LIN {X 0,Y 474.637,Z 227.855,A -85,B 0,C 180,E1 -7347.785,E2 -7347.785} C_VEL
LIN {X 0,Y 474.608,Z 227.868,A -85,B 0,C 180,E1 -7350.888,E2 -7350.888} C_VEL
LIN {X 0,Y 474.599,Z 227.864,A -85,B 0,C 180,E1 -7353.622,E2 -7353.622} C_VEL
LIN {X 0,Y 474.643,Z 227.855,A -85,B 0,C 180,E1 -7356.64,E2 -7356.64} C_VEL
LIN {X 0,Y 474.662,Z 227.851,A -85,B 0,C 180,E1 -7360.087,E2 -7360.087} C_VEL
LIN {X 0,Y 474.645,Z 227.858,A -85,B 0,C 180,E1 -7362.771,E2 -7362.771} C_VEL
LIN {X 0,Y 474.652,Z 227.858,A -85,B 0,C 180,E1 -7365.418,E2 -7365.418} C_VEL
LIN {X 0,Y 474.71,Z 227.848,A -85,B 0,C 180,E1 -7368.034,E2 -7368.034} C_VEL
LIN {X 0,Y 474.707,Z 227.853,A -85,B 0,C 180,E1 -7371.483,E2 -7371.483} C_VEL
LIN {X 0,Y 474.762,Z 227.845,A -85,B 0,C 180,E1 -7374.049,E2 -7374.049} C_VEL
LIN {X 0,Y 474.884,Z 227.829,A -85,B 0,C 180,E1 -7377.452,E2 -7377.452} C_VEL
LIN {X 0,Y 474.91,Z 227.829,A -85,B 0,C 180,E1 -7379.996,E2 -7379.996} C_VEL
LIN {X 0,Y 474.884,Z 227.825,A -85,B 0,C 180,E1 -7382.541,E2 -7382.541} C_VEL
LIN {X 0,Y 474.755,Z 227.847,A -85,B 0,C 180,E1 -7385.944,E2 -7385.944} C_VEL
LIN {X 0,Y 474.708,Z 227.856,A -85,B 0,C 180,E1 -7388.51,E2 -7388.51} C_VEL
LIN {X 0,Y 474.698,Z 227.848,A -85,B 0,C 180,E1 -7391.958,E2 -7391.958} C_VEL
LIN {X 0,Y 474.691,Z 227.848,A -85,B 0,C 180,E1 -7395.451,E2 -7395.451} C_VEL
LIN {X 0,Y 474.652,Z 227.86,A -85,B 0,C 180,E1 -7399.006,E2 -7399.006} C_VEL
LIN {X 0,Y 474.579,Z 227.863,A -85,B 0,C 180,E1 -7401.724,E2 -7401.724} C_VEL
LIN {X 0,Y 474.643,Z 227.86,A -85,B 0,C 180,E1 -7404.488,E2 -7404.488} C_VEL
LIN {X 0,Y 474.681,Z 227.856,A -85,B 0,C 180,E1 -7407.334,E2 -7407.334} C_VEL
LIN {X 0,Y 474.583,Z 227.865,A -85,B 0,C 180,E1 -7410.806,E2 -7410.806} C_VEL
LIN {X 0,Y 474.614,Z 227.86,A -85,B 0,C 180,E1 -7413.979,E2 -7413.979} C_VEL
LIN {X 0,Y 474.551,Z 227.872,A -85,B 0,C 180,E1 -7416.896,E2 -7416.896} C_VEL
LIN {X 0,Y 474.639,Z 227.864,A -85,B 0,C 180,E1 -7419.649,E2 -7419.649} C_VEL
LIN {X 0,Y 474.621,Z 227.863,A -85,B 0,C 180,E1 -7422.926,E2 -7422.926} C_VEL
LIN {X 0,Y 474.585,Z 227.871,A -85,B 0,C 180,E1 -7425.892,E2 -7425.892} C_VEL
LIN {X 0,Y 474.641,Z 227.863,A -85,B 0,C 180,E1 -7429.03,E2 -7429.03} C_VEL
LIN {X 0,Y 474.664,Z 228.034,A -85,B 0,C 180,E1 -7429.413,E2 -7429.413} C_VEL
LIN {X 0,Y 476.042,Z 236.042,A -85,B 0,C 180,E1 -7431.082,E2 -7431.082} C_VEL
LIN {X 0,Y 475.687,Z 249.987,A -85,B 0,C 180,E1 -7433.774,E2 -7433.774} C_VEL
LIN {X 0,Y 475.438,Z 257.892,A -85,B 0,C 180,E1 -7435.224,E2 -7435.224} C_VEL
LIN {X 0,Y 478.234,Z 273.822,A -85,B 0,C 180,E1 -7435.606,E2 -7435.606} C_VEL
LIN {X 0,Y 477.459,Z 365.537,A -85,B 0,C 180,E1 -7437.025,E2 -7437.025} C_VEL
LIN {X 0,Y 477.168,Z 379.142,A -85,B 0,C 180,E1 -7437.417,E2 -7437.417} C_VEL
LIN {X 0,Y 477.152,Z 379.469,A -85,B 0,C 180,E1 -7437.429,E2 -7437.429} C_VEL
LIN {X 0,Y 476.275,Z 385.106,A -85,B 0,C 180,E1 -7437.621,E2 -7437.621} C_VEL
LIN {X 0,Y 473.236,Z 394.135,A -85,B 0,C 180,E1 -7437.957,E2 -7437.957} C_VEL
LIN {X 0,Y 470.185,Z 402.828,A -85,B 0,C 180,E1 -7438.392,E2 -7438.392} C_VEL
LIN {X 0,Y 469.29,Z 407.927,A -85,B 0,C 180,E1 -7438.735,E2 -7438.735} C_VEL
LIN {X 0,Y 468.72,Z 419.724,A -85,B 0,C 180,E1 -7439.723,E2 -7439.723} C_VEL
LIN {X 0,Y 468.195,Z 430.121,A -85,B 0,C 180,E1 -7440.818,E2 -7440.818} C_VEL
LIN {X 0,Y 467.739,Z 439.1,A -85,B 0,C 180,E1 -7441.995,E2 -7441.995} C_VEL
LIN {X 0,Y 467.345,Z 446.512,A -85,B 0,C 180,E1 -7443.183,E2 -7443.183} C_VEL
LIN {X 0,Y 467.063,Z 453.262,A -85,B 0,C 180,E1 -7444.518,E2 -7444.518} C_VEL
LIN {X 0,Y 466.854,Z 459.174,A -85,B 0,C 180,E1 -7446.017,E2 -7446.017} C_VEL
LIN {X 0,Y 466.701,Z 463.326,A -85,B 0,C 180,E1 -7447.418,E2 -7447.418} C_VEL
LIN {X 0,Y 466.582,Z 466.653,A -85,B 0,C 180,E1 -7449.032,E2 -7449.032} C_VEL
LIN {X 0,Y 466.545,Z 468.549,A -85,B 0,C 180,E1 -7450.646,E2 -7450.646} C_VEL
LIN {X 0,Y 466.52,Z 468.981,A -85,B 0,C 180,E1 -7451.616,E2 -7451.616} C_VEL
LIN {X 0,Y 466.521,Z 468.971,A -85,B 0,C 180,E1 -7452.464,E2 -7452.464} C_VEL
LIN {X 0,Y 466.514,Z 468.561,A -85,B 0,C 180,E1 -7453.367,E2 -7453.367} C_VEL
LIN {X 0,Y 466.59,Z 467.307,A -85,B 0,C 180,E1 -7454.555,E2 -7454.555} C_VEL
LIN {X 0,Y 466.641,Z 464.653,A -85,B 0,C 180,E1 -7456.056,E2 -7456.056} C_VEL
LIN {X 0,Y 466.745,Z 461.18,A -85,B 0,C 180,E1 -7457.389,E2 -7457.389} C_VEL
LIN {X 0,Y 466.934,Z 456.593,A -85,B 0,C 180,E1 -7458.716,E2 -7458.716} C_VEL
LIN {X 0,Y 467.209,Z 449.631,A -85,B 0,C 180,E1 -7460.257,E2 -7460.257} C_VEL
LIN {X 0,Y 467.548,Z 442.094,A -85,B 0,C 180,E1 -7461.572,E2 -7461.572} C_VEL
LIN {X 0,Y 467.973,Z 433.15,A -85,B 0,C 180,E1 -7462.826,E2 -7462.826} C_VEL
LIN {X 0,Y 468.408,Z 422.966,A -85,B 0,C 180,E1 -7463.971,E2 -7463.971} C_VEL
LIN {X 0,Y 468.96,Z 412.135,A -85,B 0,C 180,E1 -7464.949,E2 -7464.949} C_VEL
LIN {X 0,Y 469.409,Z 401.596,A -85,B 0,C 180,E1 -7465.707,E2 -7465.707} C_VEL
LIN {X 0,Y 469.91,Z 388.899,A -85,B 0,C 180,E1 -7466.409,E2 -7466.409} C_VEL
LIN {X 0,Y 470.236,Z 376.257,A -85,B 0,C 180,E1 -7466.921,E2 -7466.921} C_VEL
LIN {X 0,Y 470.504,Z 364.115,A -85,B 0,C 180,E1 -7467.244,E2 -7467.244} C_VEL
LIN {X 0,Y 471.129,Z 273.319,A -85,B 0,C 180,E1 -7468.655,E2 -7468.655} C_VEL
LIN {X 0,Y 468.393,Z 258.274,A -85,B 0,C 180,E1 -7469.001,E2 -7469.001} C_VEL
LIN {X 0,Y 468.433,Z 255.04,A -85,B 0,C 180,E1 -7469.57,E2 -7469.57} C_VEL
LIN {X 0,Y 469.17,Z 238.914,A -85,B 0,C 180,E1 -7472.79,E2 -7472.79} C_VEL
LIN {X 0,Y 468.733,Z 234.785,A -85,B 0,C 180,E1 -7473.653,E2 -7473.653} C_VEL
LIN {X 0,Y 467.699,Z 228.785,A -85,B 0,C 180,E1 -7474.983,E2 -7474.983} C_VEL
LIN {X 0,Y 467.705,Z 228.724,A -85,B 0,C 180,E1 -7477.772,E2 -7477.772} C_VEL
LIN {X 0,Y 467.647,Z 228.73,A -85,B 0,C 180,E1 -7481.266,E2 -7481.266} C_VEL
LIN {X 0,Y 467.614,Z 228.734,A -85,B 0,C 180,E1 -7483.914,E2 -7483.914} C_VEL
LIN {X 0,Y 467.564,Z 228.745,A -85,B 0,C 180,E1 -7486.594,E2 -7486.594} C_VEL
LIN {X 0,Y 467.583,Z 228.731,A -85,B 0,C 180,E1 -7489.309,E2 -7489.309} C_VEL
LIN {X 0,Y 467.581,Z 228.736,A -85,B 0,C 180,E1 -7492.071,E2 -7492.071} C_VEL
LIN {X 0,Y 467.605,Z 228.723,A -85,B 0,C 180,E1 -7495.621,E2 -7495.621} C_VEL
LIN {X 0,Y 467.555,Z 228.732,A -85,B 0,C 180,E1 -7498.751,E2 -7498.751} C_VEL
LIN {X 0,Y 467.577,Z 228.742,A -85,B 0,C 180,E1 -7501.74,E2 -7501.74} C_VEL
LIN {X 0,Y 467.546,Z 228.738,A -85,B 0,C 180,E1 -7504.834,E2 -7504.834} C_VEL
LIN {X 0,Y 467.561,Z 228.742,A -85,B 0,C 180,E1 -7508.044,E2 -7508.044} C_VEL
LIN {X 0,Y 467.566,Z 228.737,A -85,B 0,C 180,E1 -7510.265,E2 -7510.265} C_VEL
LIN {X 0,Y 467.602,Z 228.732,A -85,B 0,C 180,E1 -7513.738,E2 -7513.738} C_VEL
LIN {X 0,Y 467.604,Z 228.738,A -85,B 0,C 180,E1 -7516.269,E2 -7516.269} C_VEL
LIN {X 0,Y 467.57,Z 228.738,A -85,B 0,C 180,E1 -7519.742,E2 -7519.742} C_VEL
LIN {X 0,Y 467.526,Z 228.738,A -85,B 0,C 180,E1 -7522.816,E2 -7522.816} C_VEL
LIN {X 0,Y 467.561,Z 228.745,A -85,B 0,C 180,E1 -7526.216,E2 -7526.216} C_VEL
LIN {X 0,Y 467.551,Z 228.736,A -85,B 0,C 180,E1 -7529.271,E2 -7529.271} C_VEL
LIN {X 0,Y 467.623,Z 228.721,A -85,B 0,C 180,E1 -7532.463,E2 -7532.463} C_VEL
LIN {X 0,Y 467.586,Z 228.735,A -85,B 0,C 180,E1 -7535.117,E2 -7535.117} C_VEL
LIN {X 0,Y 467.532,Z 228.742,A -85,B 0,C 180,E1 -7537.931,E2 -7537.931} C_VEL
LIN {X 0,Y 467.609,Z 228.737,A -85,B 0,C 180,E1 -7540.697,E2 -7540.697} C_VEL
LIN {X 0,Y 467.636,Z 228.713,A -85,B 0,C 180,E1 -7544.119,E2 -7544.119} C_VEL
LIN {X 0,Y 467.673,Z 228.721,A -85,B 0,C 180,E1 -7547.86,E2 -7547.86} C_VEL
LIN {X 0,Y 467.675,Z 228.732,A -85,B 0,C 180,E1 -7551.361,E2 -7551.361} C_VEL
LIN {X 0,Y 467.739,Z 228.713,A -85,B 0,C 180,E1 -7553.967,E2 -7553.967} C_VEL
LIN {X 0,Y 467.854,Z 228.691,A -85,B 0,C 180,E1 -7557.421,E2 -7557.421} C_VEL
LIN {X 0,Y 467.879,Z 228.697,A -85,B 0,C 180,E1 -7560.004,E2 -7560.004} C_VEL
LIN {X 0,Y 467.857,Z 228.701,A -85,B 0,C 180,E1 -7562.587,E2 -7562.587} C_VEL
LIN {X 0,Y 467.722,Z 228.722,A -85,B 0,C 180,E1 -7566.041,E2 -7566.041} C_VEL
LIN {X 0,Y 467.68,Z 228.713,A -85,B 0,C 180,E1 -7568.646,E2 -7568.646} C_VEL
LIN {X 0,Y 467.656,Z 228.728,A -85,B 0,C 180,E1 -7572.361,E2 -7572.361} C_VEL
LIN {X 0,Y 467.653,Z 228.73,A -85,B 0,C 180,E1 -7575.888,E2 -7575.888} C_VEL
LIN {X 0,Y 467.626,Z 228.724,A -85,B 0,C 180,E1 -7579.311,E2 -7579.311} C_VEL
LIN {X 0,Y 467.539,Z 228.734,A -85,B 0,C 180,E1 -7582.077,E2 -7582.077} C_VEL
LIN {X 0,Y 467.591,Z 228.741,A -85,B 0,C 180,E1 -7584.891,E2 -7584.891} C_VEL
LIN {X 0,Y 467.621,Z 228.729,A -85,B 0,C 180,E1 -7587.772,E2 -7587.772} C_VEL
LIN {X 0,Y 467.573,Z 228.74,A -85,B 0,C 180,E1 -7591.047,E2 -7591.047} C_VEL
LIN {X 0,Y 467.583,Z 228.738,A -85,B 0,C 180,E1 -7594.242,E2 -7594.242} C_VEL
LIN {X 0,Y 467.55,Z 228.742,A -85,B 0,C 180,E1 -7597.187,E2 -7597.187} C_VEL
LIN {X 0,Y 467.578,Z 228.737,A -85,B 0,C 180,E1 -7600.267,E2 -7600.267} C_VEL
LIN {X 0,Y 467.556,Z 228.729,A -85,B 0,C 180,E1 -7603.747,E2 -7603.747} C_VEL
LIN {X 0,Y 467.556,Z 228.731,A -85,B 0,C 180,E1 -7606.256,E2 -7606.256} C_VEL
LIN {X 0,Y 467.583,Z 228.736,A -85,B 0,C 180,E1 -7608.725,E2 -7608.725} C_VEL
LIN {X 0,Y 467.569,Z 228.739,A -85,B 0,C 180,E1 -7611.956,E2 -7611.956} C_VEL
LIN {X 0,Y 467.571,Z 228.739,A -85,B 0,C 180,E1 -7615.168,E2 -7615.168} C_VEL
LIN {X 0,Y 467.59,Z 228.739,A -85,B 0,C 180,E1 -7618.261,E2 -7618.261} C_VEL
LIN {X 0,Y 467.581,Z 228.739,A -85,B 0,C 180,E1 -7621.251,E2 -7621.251} C_VEL
LIN {X 0,Y 467.596,Z 228.741,A -85,B 0,C 180,E1 -7624.16,E2 -7624.16} C_VEL
LIN {X 0,Y 467.665,Z 228.954,A -85,B 0,C 180,E1 -7625.235,E2 -7625.235} C_VEL
LIN {X 0,Y 469.553,Z 239.303,A -85,B 0,C 180,E1 -7627.331,E2 -7627.331} C_VEL
LIN {X 0,Y 468.955,Z 255.135,A -85,B 0,C 180,E1 -7630.294,E2 -7630.294} C_VEL
LIN {X 0,Y 468.373,Z 270.018,A -85,B 0,C 180,E1 -7633.014,E2 -7633.014} C_VEL
LIN {X 0,Y 469.963,Z 280.323,A -85,B 0,C 180,E1 -7633.263,E2 -7633.263} C_VEL
LIN {X 0,Y 471.138,Z 288.078,A -85,B 0,C 180,E1 -7633.424,E2 -7633.424} C_VEL
LIN {X 0,Y 470.492,Z 377.726,A -85,B 0,C 180,E1 -7634.819,E2 -7634.819} C_VEL
LIN {X 0,Y 470.152,Z 391.02,A -85,B 0,C 180,E1 -7635.196,E2 -7635.196} C_VEL
LIN {X 0,Y 469.722,Z 403.201,A -85,B 0,C 180,E1 -7635.708,E2 -7635.708} C_VEL
LIN {X 0,Y 469.256,Z 415.01,A -85,B 0,C 180,E1 -7636.379,E2 -7636.379} C_VEL
LIN {X 0,Y 468.786,Z 426.018,A -85,B 0,C 180,E1 -7637.188,E2 -7637.188} C_VEL
LIN {X 0,Y 468.288,Z 437.008,A -85,B 0,C 180,E1 -7638.201,E2 -7638.201} C_VEL
LIN {X 0,Y 467.837,Z 445.632,A -85,B 0,C 180,E1 -7639.177,E2 -7639.177} C_VEL
LIN {X 0,Y 467.483,Z 453.579,A -85,B 0,C 180,E1 -7640.263,E2 -7640.263} C_VEL
LIN {X 0,Y 467.155,Z 461.345,A -85,B 0,C 180,E1 -7641.566,E2 -7641.566} C_VEL
LIN {X 0,Y 466.861,Z 468.474,A -85,B 0,C 180,E1 -7643.083,E2 -7643.083} C_VEL
LIN {X 0,Y 466.792,Z 473.223,A -85,B 0,C 180,E1 -7644.384,E2 -7644.384} C_VEL
LIN {X 0,Y 466.65,Z 476.849,A -85,B 0,C 180,E1 -7645.682,E2 -7645.682} C_VEL
LIN {X 0,Y 466.663,Z 478.724,A -85,B 0,C 180,E1 -7646.547,E2 -7646.547} C_VEL
LIN {X 0,Y 466.647,Z 480.131,A -85,B 0,C 180,E1 -7647.411,E2 -7647.411} C_VEL
LIN {X 0,Y 466.592,Z 481.746,A -85,B 0,C 180,E1 -7649.137,E2 -7649.137} C_VEL
LIN {X 0,Y 466.601,Z 481.972,A -85,B 0,C 180,E1 -7650,E2 -7650} C_VEL
LIN {X 0,Y 466.592,Z 481.767,A -85,B 0,C 180,E1 -7650.863,E2 -7650.863} C_VEL
LIN {X 0,Y 466.647,Z 480.18,A -85,B 0,C 180,E1 -7652.59,E2 -7652.59} C_VEL
LIN {X 0,Y 466.664,Z 478.797,A -85,B 0,C 180,E1 -7653.454,E2 -7653.454} C_VEL
LIN {X 0,Y 466.694,Z 475.879,A -85,B 0,C 180,E1 -7654.751,E2 -7654.751} C_VEL
LIN {X 0,Y 466.782,Z 471.931,A -85,B 0,C 180,E1 -7656.05,E2 -7656.05} C_VEL
LIN {X 0,Y 466.948,Z 466.852,A -85,B 0,C 180,E1 -7657.35,E2 -7657.35} C_VEL
LIN {X 0,Y 467.215,Z 460.46,A -85,B 0,C 180,E1 -7658.652,E2 -7658.652} C_VEL
LIN {X 0,Y 467.591,Z 452.478,A -85,B 0,C 180,E1 -7659.954,E2 -7659.954} C_VEL
LIN {X 0,Y 467.945,Z 444.35,A -85,B 0,C 180,E1 -7661.04,E2 -7661.04} C_VEL
LIN {X 0,Y 468.501,Z 434.442,A -85,B 0,C 180,E1 -7662.123,E2 -7662.123} C_VEL
LIN {X 0,Y 468.916,Z 424.151,A -85,B 0,C 180,E1 -7663.037,E2 -7663.037} C_VEL
LIN {X 0,Y 469.503,Z 412.408,A -85,B 0,C 180,E1 -7663.857,E2 -7663.857} C_VEL
LIN {X 0,Y 469.975,Z 400.378,A -85,B 0,C 180,E1 -7664.506,E2 -7664.506} C_VEL
LIN {X 0,Y 470.379,Z 388.034,A -85,B 0,C 180,E1 -7664.991,E2 -7664.991} C_VEL
LIN {X 0,Y 470.692,Z 375.29,A -85,B 0,C 180,E1 -7665.313,E2 -7665.313} C_VEL
LIN {X 0,Y 471.424,Z 287.468,A -85,B 0,C 180,E1 -7666.683,E2 -7666.683} C_VEL
LIN {X 0,Y 468.448,Z 269.998,A -85,B 0,C 180,E1 -7667.11,E2 -7667.11} C_VEL
LIN {X 0,Y 468.967,Z 255.717,A -85,B 0,C 180,E1 -7669.706,E2 -7669.706} C_VEL
LIN {X 0,Y 469.694,Z 240.012,A -85,B 0,C 180,E1 -7672.662,E2 -7672.662} C_VEL
LIN {X 0,Y 467.668,Z 229.005,A -85,B 0,C 180,E1 -7674.936,E2 -7674.936} C_VEL
LIN {X 0,Y 467.595,Z 228.743,A -85,B 0,C 180,E1 -7675.6,E2 -7675.6} C_VEL
LIN {X 0,Y 467.626,Z 228.737,A -85,B 0,C 180,E1 -7677.769,E2 -7677.769} C_VEL
LIN {X 0,Y 467.577,Z 228.737,A -85,B 0,C 180,E1 -7681.044,E2 -7681.044} C_VEL
LIN {X 0,Y 467.599,Z 228.741,A -85,B 0,C 180,E1 -7684.241,E2 -7684.241} C_VEL
LIN {X 0,Y 467.553,Z 228.742,A -85,B 0,C 180,E1 -7687.184,E2 -7687.184} C_VEL
LIN {X 0,Y 467.57,Z 228.745,A -85,B 0,C 180,E1 -7690.265,E2 -7690.265} C_VEL
LIN {X 0,Y 467.572,Z 228.737,A -85,B 0,C 180,E1 -7692.562,E2 -7692.562} C_VEL
LIN {X 0,Y 467.576,Z 228.739,A -85,B 0,C 180,E1 -7695.051,E2 -7695.051} C_VEL
LIN {X 0,Y 467.584,Z 228.737,A -85,B 0,C 180,E1 -7698.595,E2 -7698.595} C_VEL
LIN {X 0,Y 467.572,Z 228.736,A -85,B 0,C 180,E1 -7701.953,E2 -7701.953} C_VEL
LIN {X 0,Y 467.566,Z 228.743,A -85,B 0,C 180,E1 -7705.165,E2 -7705.165} C_VEL
LIN {X 0,Y 467.588,Z 228.734,A -85,B 0,C 180,E1 -7708.257,E2 -7708.257} C_VEL
LIN {X 0,Y 467.554,Z 228.742,A -85,B 0,C 180,E1 -7711.246,E2 -7711.246} C_VEL
LIN {X 0,Y 467.587,Z 228.736,A -85,B 0,C 180,E1 -7714.399,E2 -7714.399} C_VEL
LIN {X 0,Y 467.581,Z 228.739,A -85,B 0,C 180,E1 -7716.993,E2 -7716.993} C_VEL
LIN {X 0,Y 467.63,Z 228.729,A -85,B 0,C 180,E1 -7719.774,E2 -7719.774} C_VEL
LIN {X 0,Y 467.605,Z 228.734,A -85,B 0,C 180,E1 -7722.503,E2 -7722.503} C_VEL
LIN {X 0,Y 467.61,Z 228.732,A -85,B 0,C 180,E1 -7725.193,E2 -7725.193} C_VEL
LIN {X 0,Y 467.662,Z 228.728,A -85,B 0,C 180,E1 -7727.851,E2 -7727.851} C_VEL
LIN {X 0,Y 467.666,Z 228.729,A -85,B 0,C 180,E1 -7731.353,E2 -7731.353} C_VEL
LIN {X 0,Y 467.727,Z 228.721,A -85,B 0,C 180,E1 -7733.959,E2 -7733.959} C_VEL
LIN {X 0,Y 467.848,Z 228.705,A -85,B 0,C 180,E1 -7737.413,E2 -7737.413} C_VEL
LIN {X 0,Y 467.88,Z 228.704,A -85,B 0,C 180,E1 -7739.996,E2 -7739.996} C_VEL
LIN {X 0,Y 467.849,Z 228.701,A -85,B 0,C 180,E1 -7742.579,E2 -7742.579} C_VEL
LIN {X 0,Y 467.718,Z 228.725,A -85,B 0,C 180,E1 -7746.034,E2 -7746.034} C_VEL
LIN {X 0,Y 467.665,Z 228.731,A -85,B 0,C 180,E1 -7748.639,E2 -7748.639} C_VEL
LIN {X 0,Y 467.649,Z 228.728,A -85,B 0,C 180,E1 -7752.141,E2 -7752.141} C_VEL
LIN {X 0,Y 467.63,Z 228.728,A -85,B 0,C 180,E1 -7755.691,E2 -7755.691} C_VEL
LIN {X 0,Y 467.611,Z 228.734,A -85,B 0,C 180,E1 -7759.303,E2 -7759.303} C_VEL
LIN {X 0,Y 467.524,Z 228.742,A -85,B 0,C 180,E1 -7762.069,E2 -7762.069} C_VEL
LIN {X 0,Y 467.588,Z 228.737,A -85,B 0,C 180,E1 -7764.883,E2 -7764.883} C_VEL
LIN {X 0,Y 467.609,Z 228.734,A -85,B 0,C 180,E1 -7767.764,E2 -7767.764} C_VEL
LIN {X 0,Y 467.547,Z 228.74,A -85,B 0,C 180,E1 -7771.04,E2 -7771.04} C_VEL
LIN {X 0,Y 467.566,Z 228.737,A -85,B 0,C 180,E1 -7774.238,E2 -7774.238} C_VEL
LIN {X 0,Y 467.526,Z 228.751,A -85,B 0,C 180,E1 -7777.183,E2 -7777.183} C_VEL
LIN {X 0,Y 467.573,Z 228.738,A -85,B 0,C 180,E1 -7780.258,E2 -7780.258} C_VEL
LIN {X 0,Y 467.589,Z 228.738,A -85,B 0,C 180,E1 -7782.567,E2 -7782.567} C_VEL
LIN {X 0,Y 467.541,Z 228.746,A -85,B 0,C 180,E1 -7786.172,E2 -7786.172} C_VEL
LIN {X 0,Y 467.628,Z 228.872,A -85,B 0,C 180,E1 -7789.174,E2 -7789.174} C_VEL
LIN {X 0,Y 469.008,Z 236.06,A -85,B 0,C 180,E1 -7790.72,E2 -7790.72} C_VEL
LIN {X 0,Y 469.017,Z 242.983,A -85,B 0,C 180,E1 -7792.094,E2 -7792.094} C_VEL
LIN {X 0,Y 468.516,Z 257.651,A -85,B 0,C 180,E1 -7794.905,E2 -7794.905} C_VEL
LIN {X 0,Y 468.727,Z 259.266,A -85,B 0,C 180,E1 -7794.995,E2 -7794.995} C_VEL
LIN {X 0,Y 471.45,Z 273.753,A -85,B 0,C 180,E1 -7795.34,E2 -7795.34} C_VEL
LIN {X 0,Y 470.64,Z 365.96,A -85,B 0,C 180,E1 -7796.794,E2 -7796.794} C_VEL
LIN {X 0,Y 470.313,Z 379.843,A -85,B 0,C 180,E1 -7797.205,E2 -7797.205} C_VEL
LIN {X 0,Y 469.915,Z 392.024,A -85,B 0,C 180,E1 -7797.741,E2 -7797.741} C_VEL
LIN {X 0,Y 469.456,Z 404.486,A -85,B 0,C 180,E1 -7798.492,E2 -7798.492} C_VEL
LIN {X 0,Y 469.29,Z 407.927,A -85,B 0,C 180,E1 -7798.735,E2 -7798.735} C_VEL
LIN {X 0,Y 468.44,Z 411.387,A -85,B 0,C 180,E1 -7798.976,E2 -7798.976} C_VEL
LIN {X 0,Y 462.33,Z 421.783,A -85,B 0,C 180,E1 -7799.726,E2 -7799.726} C_VEL
LIN {X 0,Y 461.536,Z 424.803,A -85,B 0,C 180,E1 -7800.018,E2 -7800.018} C_VEL
LIN {X 0,Y 461.063,Z 433.66,A -85,B 0,C 180,E1 -7801.055,E2 -7801.055} C_VEL
LIN {X 0,Y 460.598,Z 441.92,A -85,B 0,C 180,E1 -7802.236,E2 -7802.236} C_VEL
LIN {X 0,Y 460.19,Z 448.957,A -85,B 0,C 180,E1 -7803.467,E2 -7803.467} C_VEL
LIN {X 0,Y 459.959,Z 454.575,A -85,B 0,C 180,E1 -7804.67,E2 -7804.67} C_VEL
LIN {X 0,Y 459.76,Z 459.893,A -85,B 0,C 180,E1 -7806.104,E2 -7806.104} C_VEL
LIN {X 0,Y 459.595,Z 463.883,A -85,B 0,C 180,E1 -7807.524,E2 -7807.524} C_VEL
LIN {X 0,Y 459.503,Z 466.609,A -85,B 0,C 180,E1 -7808.887,E2 -7808.887} C_VEL
LIN {X 0,Y 459.468,Z 468.407,A -85,B 0,C 180,E1 -7810.335,E2 -7810.335} C_VEL
LIN {X 0,Y 459.435,Z 469.061,A -85,B 0,C 180,E1 -7811.496,E2 -7811.496} C_VEL
LIN {X 0,Y 459.421,Z 468.809,A -85,B 0,C 180,E1 -7813.103,E2 -7813.103} C_VEL
LIN {X 0,Y 459.494,Z 467.551,A -85,B 0,C 180,E1 -7814.467,E2 -7814.467} C_VEL
LIN {X 0,Y 459.571,Z 464.344,A -85,B 0,C 180,E1 -7816.288,E2 -7816.288} C_VEL
LIN {X 0,Y 459.711,Z 460.721,A -85,B 0,C 180,E1 -7817.641,E2 -7817.641} C_VEL
LIN {X 0,Y 459.906,Z 455.962,A -85,B 0,C 180,E1 -7818.988,E2 -7818.988} C_VEL
LIN {X 0,Y 460.178,Z 448.815,A -85,B 0,C 180,E1 -7820.55,E2 -7820.55} C_VEL
LIN {X 0,Y 460.565,Z 441.051,A -85,B 0,C 180,E1 -7821.885,E2 -7821.885} C_VEL
LIN {X 0,Y 460.952,Z 433.107,A -85,B 0,C 180,E1 -7822.994,E2 -7822.994} C_VEL
LIN {X 0,Y 461.423,Z 423.429,A -85,B 0,C 180,E1 -7824.099,E2 -7824.099} C_VEL
LIN {X 0,Y 461.986,Z 412.667,A -85,B 0,C 180,E1 -7825.091,E2 -7825.091} C_VEL
LIN {X 0,Y 462.459,Z 402.248,A -85,B 0,C 180,E1 -7825.86,E2 -7825.86} C_VEL
LIN {X 0,Y 462.963,Z 389.721,A -85,B 0,C 180,E1 -7826.573,E2 -7826.573} C_VEL
LIN {X 0,Y 463.342,Z 376.536,A -85,B 0,C 180,E1 -7827.12,E2 -7827.12} C_VEL
LIN {X 0,Y 463.621,Z 364.26,A -85,B 0,C 180,E1 -7827.453,E2 -7827.453} C_VEL
LIN {X 0,Y 464.323,Z 274.391,A -85,B 0,C 180,E1 -7828.867,E2 -7828.867} C_VEL
LIN {X 0,Y 461.422,Z 258.56,A -85,B 0,C 180,E1 -7829.236,E2 -7829.236} C_VEL
LIN {X 0,Y 461.376,Z 257.565,A -85,B 0,C 180,E1 -7829.345,E2 -7829.345} C_VEL
LIN {X 0,Y 462.078,Z 242.394,A -85,B 0,C 180,E1 -7832.397,E2 -7832.397} C_VEL
LIN {X 0,Y 462.129,Z 238.148,A -85,B 0,C 180,E1 -7833.269,E2 -7833.269} C_VEL
LIN {X 0,Y 460.675,Z 229.686,A -85,B 0,C 180,E1 -7835.142,E2 -7835.142} C_VEL
LIN {X 0,Y 460.651,Z 229.604,A -85,B 0,C 180,E1 -7837.892,E2 -7837.892} C_VEL
LIN {X 0,Y 460.623,Z 229.605,A -85,B 0,C 180,E1 -7841.44,E2 -7841.44} C_VEL
LIN {X 0,Y 460.572,Z 229.613,A -85,B 0,C 180,E1 -7844.131,E2 -7844.131} C_VEL
LIN {X 0,Y 460.53,Z 229.62,A -85,B 0,C 180,E1 -7846.855,E2 -7846.855} C_VEL
LIN {X 0,Y 460.53,Z 229.607,A -85,B 0,C 180,E1 -7849.617,E2 -7849.617} C_VEL
LIN {X 0,Y 460.53,Z 229.616,A -85,B 0,C 180,E1 -7852.427,E2 -7852.427} C_VEL
LIN {X 0,Y 460.54,Z 229.601,A -85,B 0,C 180,E1 -7855.809,E2 -7855.809} C_VEL
LIN {X 0,Y 460.522,Z 229.605,A -85,B 0,C 180,E1 -7858.234,E2 -7858.234} C_VEL
LIN {X 0,Y 460.542,Z 229.62,A -85,B 0,C 180,E1 -7861.299,E2 -7861.299} C_VEL
LIN {X 0,Y 460.534,Z 229.61,A -85,B 0,C 180,E1 -7864.517,E2 -7864.517} C_VEL
LIN {X 0,Y 460.505,Z 229.625,A -85,B 0,C 180,E1 -7867.622,E2 -7867.622} C_VEL
LIN {X 0,Y 460.528,Z 229.613,A -85,B 0,C 180,E1 -7870.277,E2 -7870.277} C_VEL
LIN {X 0,Y 460.53,Z 229.608,A -85,B 0,C 180,E1 -7873.371,E2 -7873.371} C_VEL
LIN {X 0,Y 460.532,Z 229.615,A -85,B 0,C 180,E1 -7876.636,E2 -7876.636} C_VEL
LIN {X 0,Y 460.553,Z 229.607,A -85,B 0,C 180,E1 -7880.147,E2 -7880.147} C_VEL
LIN {X 0,Y 460.454,Z 229.618,A -85,B 0,C 180,E1 -7883.475,E2 -7883.475} C_VEL
LIN {X 0,Y 460.503,Z 229.622,A -85,B 0,C 180,E1 -7886.68,E2 -7886.68} C_VEL
LIN {X 0,Y 460.503,Z 229.614,A -85,B 0,C 180,E1 -7889.766,E2 -7889.766} C_VEL
LIN {X 0,Y 460.562,Z 229.601,A -85,B 0,C 180,E1 -7892.761,E2 -7892.761} C_VEL
LIN {X 0,Y 460.525,Z 229.611,A -85,B 0,C 180,E1 -7895.672,E2 -7895.672} C_VEL
LIN {X 0,Y 460.536,Z 229.619,A -85,B 0,C 180,E1 -7898.572,E2 -7898.572} C_VEL
LIN {X 0,Y 460.576,Z 229.606,A -85,B 0,C 180,E1 -7901.315,E2 -7901.315} C_VEL
LIN {X 0,Y 460.59,Z 229.59,A -85,B 0,C 180,E1 -7904.063,E2 -7904.063} C_VEL
LIN {X 0,Y 460.619,Z 229.601,A -85,B 0,C 180,E1 -7907.671,E2 -7907.671} C_VEL
LIN {X 0,Y 460.622,Z 229.61,A -85,B 0,C 180,E1 -7911.228,E2 -7911.228} C_VEL
LIN {X 0,Y 460.705,Z 229.59,A -85,B 0,C 180,E1 -7913.874,E2 -7913.874} C_VEL
LIN {X 0,Y 460.795,Z 229.57,A -85,B 0,C 180,E1 -7917.382,E2 -7917.382} C_VEL
LIN {X 0,Y 460.849,Z 229.572,A -85,B 0,C 180,E1 -7920.004,E2 -7920.004} C_VEL
LIN {X 0,Y 460.798,Z 229.58,A -85,B 0,C 180,E1 -7922.626,E2 -7922.626} C_VEL
LIN {X 0,Y 460.686,Z 229.597,A -85,B 0,C 180,E1 -7926.134,E2 -7926.134} C_VEL
LIN {X 0,Y 460.627,Z 229.591,A -85,B 0,C 180,E1 -7928.78,E2 -7928.78} C_VEL
LIN {X 0,Y 460.616,Z 229.604,A -85,B 0,C 180,E1 -7932.448,E2 -7932.448} C_VEL
LIN {X 0,Y 460.604,Z 229.609,A -85,B 0,C 180,E1 -7936.001,E2 -7936.001} C_VEL
LIN {X 0,Y 460.572,Z 229.602,A -85,B 0,C 180,E1 -7939.619,E2 -7939.619} C_VEL
LIN {X 0,Y 460.516,Z 229.613,A -85,B 0,C 180,E1 -7942.432,E2 -7942.432} C_VEL
LIN {X 0,Y 460.553,Z 229.612,A -85,B 0,C 180,E1 -7945.799,E2 -7945.799} C_VEL
LIN {X 0,Y 460.555,Z 229.611,A -85,B 0,C 180,E1 -7948.236,E2 -7948.236} C_VEL
LIN {X 0,Y 460.527,Z 229.618,A -85,B 0,C 180,E1 -7951.285,E2 -7951.285} C_VEL
LIN {X 0,Y 460.529,Z 229.618,A -85,B 0,C 180,E1 -7954.506,E2 -7954.506} C_VEL
LIN {X 0,Y 460.506,Z 229.617,A -85,B 0,C 180,E1 -7957.626,E2 -7957.626} C_VEL
LIN {X 0,Y 460.535,Z 229.619,A -85,B 0,C 180,E1 -7961.014,E2 -7961.014} C_VEL
LIN {X 0,Y 460.52,Z 229.601,A -85,B 0,C 180,E1 -7964.591,E2 -7964.591} C_VEL
LIN {X 0,Y 460.512,Z 229.622,A -85,B 0,C 180,E1 -7967.818,E2 -7967.818} C_VEL
LIN {X 0,Y 460.526,Z 229.616,A -85,B 0,C 180,E1 -7970.138,E2 -7970.138} C_VEL
LIN {X 0,Y 460.48,Z 229.623,A -85,B 0,C 180,E1 -7973.472,E2 -7973.472} C_VEL
LIN {X 0,Y 460.536,Z 229.616,A -85,B 0,C 180,E1 -7976.676,E2 -7976.676} C_VEL
LIN {X 0,Y 460.517,Z 229.623,A -85,B 0,C 180,E1 -7979.761,E2 -7979.761} C_VEL
LIN {X 0,Y 460.567,Z 229.616,A -85,B 0,C 180,E1 -7982.756,E2 -7982.756} C_VEL
LIN {X 0,Y 460.589,Z 229.728,A -85,B 0,C 180,E1 -7985.009,E2 -7985.009} C_VEL
LIN {X 0,Y 462.568,Z 240.293,A -85,B 0,C 180,E1 -7987.206,E2 -7987.206} C_VEL
LIN {X 0,Y 461.996,Z 254.92,A -85,B 0,C 180,E1 -7989.985,E2 -7989.985} C_VEL
LIN {X 0,Y 461.353,Z 270.009,A -85,B 0,C 180,E1 -7992.776,E2 -7992.776} C_VEL
LIN {X 0,Y 464.296,Z 288.422,A -85,B 0,C 180,E1 -7993.197,E2 -7993.197} C_VEL
LIN {X 0,Y 463.599,Z 377.961,A -85,B 0,C 180,E1 -7994.616,E2 -7994.616} C_VEL
LIN {X 0,Y 463.239,Z 391.154,A -85,B 0,C 180,E1 -7994.998,E2 -7994.998} C_VEL
LIN {X 0,Y 462.792,Z 403.856,A -85,B 0,C 180,E1 -7995.545,E2 -7995.545} C_VEL
LIN {X 0,Y 462.271,Z 415.932,A -85,B 0,C 180,E1 -7996.258,E2 -7996.258} C_VEL
LIN {X 0,Y 461.804,Z 426.59,A -85,B 0,C 180,E1 -7997.066,E2 -7997.066} C_VEL
LIN {X 0,Y 461.328,Z 436.76,A -85,B 0,C 180,E1 -7998.021,E2 -7998.021} C_VEL
LIN {X 0,Y 460.832,Z 445.417,A -85,B 0,C 180,E1 -7999.011,E2 -7999.011} C_VEL
LIN {X 0,Y 460.472,Z 453.389,A -85,B 0,C 180,E1 -8000.113,E2 -8000.113} C_VEL
LIN {X 0,Y 460.119,Z 461.179,A -85,B 0,C 180,E1 -8001.436,E2 -8001.436} C_VEL
LIN {X 0,Y 459.781,Z 468.321,A -85,B 0,C 180,E1 -8002.976,E2 -8002.976} C_VEL
LIN {X 0,Y 459.69,Z 473.082,A -85,B 0,C 180,E1 -8004.297,E2 -8004.297} C_VEL
LIN {X 0,Y 459.568,Z 476.72,A -85,B 0,C 180,E1 -8005.615,E2 -8005.615} C_VEL
LIN {X 0,Y 459.56,Z 478.6,A -85,B 0,C 180,E1 -8006.493,E2 -8006.493} C_VEL
LIN {X 0,Y 459.569,Z 480.017,A -85,B 0,C 180,E1 -8007.371,E2 -8007.371} C_VEL
LIN {X 0,Y 459.497,Z 481.641,A -85,B 0,C 180,E1 -8009.124,E2 -8009.124} C_VEL
LIN {X 0,Y 459.504,Z 481.873,A -85,B 0,C 180,E1 -8010,E2 -8010} C_VEL
LIN {X 0,Y 459.497,Z 481.675,A -85,B 0,C 180,E1 -8010.877,E2 -8010.877} C_VEL
LIN {X 0,Y 459.57,Z 480.096,A -85,B 0,C 180,E1 -8012.63,E2 -8012.63} C_VEL
LIN {X 0,Y 459.56,Z 478.718,A -85,B 0,C 180,E1 -8013.507,E2 -8013.507} C_VEL
LIN {X 0,Y 459.626,Z 475.808,A -85,B 0,C 180,E1 -8014.824,E2 -8014.824} C_VEL
LIN {X 0,Y 459.707,Z 471.868,A -85,B 0,C 180,E1 -8016.144,E2 -8016.144} C_VEL
LIN {X 0,Y 459.874,Z 466.8,A -85,B 0,C 180,E1 -8017.464,E2 -8017.464} C_VEL
LIN {X 0,Y 460.179,Z 460.433,A -85,B 0,C 180,E1 -8018.785,E2 -8018.785} C_VEL
LIN {X 0,Y 460.59,Z 452.478,A -85,B 0,C 180,E1 -8020.107,E2 -8020.107} C_VEL
LIN {X 0,Y 460.974,Z 444.383,A -85,B 0,C 180,E1 -8021.209,E2 -8021.209} C_VEL
LIN {X 0,Y 461.549,Z 434.516,A -85,B 0,C 180,E1 -8022.309,E2 -8022.309} C_VEL
LIN {X 0,Y 462.015,Z 423.449,A -85,B 0,C 180,E1 -8023.302,E2 -8023.302} C_VEL
LIN {X 0,Y 462.627,Z 412.61,A -85,B 0,C 180,E1 -8024.068,E2 -8024.068} C_VEL
LIN {X 0,Y 463.127,Z 400.664,A -85,B 0,C 180,E1 -8024.725,E2 -8024.725} C_VEL
LIN {X 0,Y 463.582,Z 387.657,A -85,B 0,C 180,E1 -8025.245,E2 -8025.245} C_VEL
LIN {X 0,Y 463.908,Z 374.728,A -85,B 0,C 180,E1 -8025.571,E2 -8025.571} C_VEL
LIN {X 0,Y 464.538,Z 287.514,A -85,B 0,C 180,E1 -8026.956,E2 -8026.956} C_VEL
LIN {X 0,Y 461.51,Z 270.075,A -85,B 0,C 180,E1 -8027.389,E2 -8027.389} C_VEL
LIN {X 0,Y 461.542,Z 267.836,A -85,B 0,C 180,E1 -8027.731,E2 -8027.731} C_VEL
LIN {X 0,Y 462.369,Z 249.717,A -85,B 0,C 180,E1 -8031.162,E2 -8031.162} C_VEL
LIN {X 0,Y 462.751,Z 241.265,A -85,B 0,C 180,E1 -8032.786,E2 -8032.786} C_VEL
LIN {X 0,Y 460.72,Z 230.436,A -85,B 0,C 180,E1 -8035.044,E2 -8035.044} C_VEL
LIN {X 0,Y 460.565,Z 229.644,A -85,B 0,C 180,E1 -8035.294,E2 -8035.294} C_VEL
LIN {X 0,Y 460.56,Z 229.617,A -85,B 0,C 180,E1 -8038.233,E2 -8038.233} C_VEL
LIN {X 0,Y 460.532,Z 229.615,A -85,B 0,C 180,E1 -8041.282,E2 -8041.282} C_VEL
LIN {X 0,Y 460.542,Z 229.617,A -85,B 0,C 180,E1 -8044.504,E2 -8044.504} C_VEL
LIN {X 0,Y 460.509,Z 229.621,A -85,B 0,C 180,E1 -8047.623,E2 -8047.623} C_VEL
LIN {X 0,Y 460.531,Z 229.616,A -85,B 0,C 180,E1 -8051.011,E2 -8051.011} C_VEL
LIN {X 0,Y 460.516,Z 229.619,A -85,B 0,C 180,E1 -8054.167,E2 -8054.167} C_VEL
LIN {X 0,Y 460.503,Z 229.61,A -85,B 0,C 180,E1 -8057.101,E2 -8057.101} C_VEL
LIN {X 0,Y 460.529,Z 229.618,A -85,B 0,C 180,E1 -8060.134,E2 -8060.134} C_VEL
LIN {X 0,Y 460.483,Z 229.622,A -85,B 0,C 180,E1 -8063.468,E2 -8063.468} C_VEL
LIN {X 0,Y 460.527,Z 229.622,A -85,B 0,C 180,E1 -8066.672,E2 -8066.672} C_VEL
LIN {X 0,Y 460.514,Z 229.618,A -85,B 0,C 180,E1 -8069.757,E2 -8069.757} C_VEL
LIN {X 0,Y 460.501,Z 229.619,A -85,B 0,C 180,E1 -8072.749,E2 -8072.749} C_VEL
LIN {X 0,Y 460.527,Z 229.614,A -85,B 0,C 180,E1 -8075.664,E2 -8075.664} C_VEL
LIN {X 0,Y 460.53,Z 229.616,A -85,B 0,C 180,E1 -8078.576,E2 -8078.576} C_VEL
LIN {X 0,Y 460.594,Z 229.611,A -85,B 0,C 180,E1 -8081.308,E2 -8081.308} C_VEL
LIN {X 0,Y 460.612,Z 229.601,A -85,B 0,C 180,E1 -8084.056,E2 -8084.056} C_VEL
LIN {X 0,Y 460.615,Z 229.609,A -85,B 0,C 180,E1 -8087.663,E2 -8087.663} C_VEL
LIN {X 0,Y 460.617,Z 229.606,A -85,B 0,C 180,E1 -8091.22,E2 -8091.22} C_VEL
LIN {X 0,Y 460.693,Z 229.596,A -85,B 0,C 180,E1 -8093.866,E2 -8093.866} C_VEL
LIN {X 0,Y 460.789,Z 229.584,A -85,B 0,C 180,E1 -8097.374,E2 -8097.374} C_VEL
LIN {X 0,Y 460.85,Z 229.58,A -85,B 0,C 180,E1 -8099.996,E2 -8099.996} C_VEL
LIN {X 0,Y 460.79,Z 229.58,A -85,B 0,C 180,E1 -8102.618,E2 -8102.618} C_VEL
LIN {X 0,Y 460.682,Z 229.603,A -85,B 0,C 180,E1 -8106.126,E2 -8106.126} C_VEL
LIN {X 0,Y 460.615,Z 229.608,A -85,B 0,C 180,E1 -8108.772,E2 -8108.772} C_VEL
LIN {X 0,Y 460.607,Z 229.609,A -85,B 0,C 180,E1 -8112.44,E2 -8112.44} C_VEL
LIN {X 0,Y 460.591,Z 229.606,A -85,B 0,C 180,E1 -8115.993,E2 -8115.993} C_VEL
LIN {X 0,Y 460.557,Z 229.612,A -85,B 0,C 180,E1 -8119.611,E2 -8119.611} C_VEL
LIN {X 0,Y 460.499,Z 229.62,A -85,B 0,C 180,E1 -8122.424,E2 -8122.424} C_VEL
LIN {X 0,Y 460.551,Z 229.603,A -85,B 0,C 180,E1 -8125.797,E2 -8125.797} C_VEL
LIN {X 0,Y 460.537,Z 229.614,A -85,B 0,C 180,E1 -8128.228,E2 -8128.228} C_VEL
LIN {X 0,Y 460.499,Z 229.618,A -85,B 0,C 180,E1 -8131.278,E2 -8131.278} C_VEL
LIN {X 0,Y 460.51,Z 229.617,A -85,B 0,C 180,E1 -8134.501,E2 -8134.501} C_VEL
LIN {X 0,Y 460.505,Z 229.619,A -85,B 0,C 180,E1 -8137.616,E2 -8137.616} C_VEL
LIN {X 0,Y 460.536,Z 229.615,A -85,B 0,C 180,E1 -8140.268,E2 -8140.268} C_VEL
LIN {X 0,Y 460.494,Z 229.623,A -85,B 0,C 180,E1 -8143.368,E2 -8143.368} C_VEL
LIN {X 0,Y 460.491,Z 229.623,A -85,B 0,C 180,E1 -8146.623,E2 -8146.623} C_VEL
LIN {X 0,Y 460.567,Z 229.73,A -85,B 0,C 180,E1 -8148.932,E2 -8148.932} C_VEL
LIN {X 0,Y 462.175,Z 238.492,A -85,B 0,C 180,E1 -8150.843,E2 -8150.843} C_VEL
LIN {X 0,Y 461.838,Z 250.99,A -85,B 0,C 180,E1 -8153.324,E2 -8153.324} C_VEL
LIN {X 0,Y 461.601,Z 257.901,A -85,B 0,C 180,E1 -8154.634,E2 -8154.634} C_VEL
LIN {X 0,Y 462.262,Z 261.53,A -85,B 0,C 180,E1 -8154.766,E2 -8154.766} C_VEL
LIN {X 0,Y 464.73,Z 275.771,A -85,B 0,C 180,E1 -8155.101,E2 -8155.101} C_VEL
LIN {X 0,Y 463.887,Z 365.482,A -85,B 0,C 180,E1 -8156.532,E2 -8156.532} C_VEL
LIN {X 0,Y 463.558,Z 378.763,A -85,B 0,C 180,E1 -8156.921,E2 -8156.921} C_VEL
LIN {X 0,Y 463.108,Z 391.334,A -85,B 0,C 180,E1 -8157.467,E2 -8157.467} C_VEL
LIN {X 0,Y 462.64,Z 402.82,A -85,B 0,C 180,E1 -8158.143,E2 -8158.143} C_VEL
LIN {X 0,Y 462.137,Z 413.991,A -85,B 0,C 180,E1 -8158.992,E2 -8158.992} C_VEL
LIN {X 0,Y 461.536,Z 424.803,A -85,B 0,C 180,E1 -8160.018,E2 -8160.018} C_VEL
LIN {X 0,Y 460.69,Z 429.26,A -85,B 0,C 180,E1 -8160.489,E2 -8160.489} C_VEL
LIN {X 0,Y 457.482,Z 436.172,A -85,B 0,C 180,E1 -8161.283,E2 -8161.283} C_VEL
LIN {X 0,Y 454.25,Z 442.491,A -85,B 0,C 180,E1 -8162.156,E2 -8162.156} C_VEL
LIN {X 0,Y 453.376,Z 446.019,A -85,B 0,C 180,E1 -8162.745,E2 -8162.745} C_VEL
LIN {X 0,Y 452.964,Z 453.469,A -85,B 0,C 180,E1 -8164.25,E2 -8164.25} C_VEL
LIN {X 0,Y 452.73,Z 459.094,A -85,B 0,C 180,E1 -8165.709,E2 -8165.709} C_VEL
LIN {X 0,Y 452.565,Z 463.319,A -85,B 0,C 180,E1 -8167.155,E2 -8167.155} C_VEL
LIN {X 0,Y 452.418,Z 466.581,A -85,B 0,C 180,E1 -8168.74,E2 -8168.74} C_VEL
LIN {X 0,Y 452.36,Z 468.258,A -85,B 0,C 180,E1 -8170.013,E2 -8170.013} C_VEL
LIN {X 0,Y 452.356,Z 469.142,A -85,B 0,C 180,E1 -8171.371,E2 -8171.371} C_VEL
LIN {X 0,Y 452.308,Z 469.056,A -85,B 0,C 180,E1 -8172.829,E2 -8172.829} C_VEL
LIN {X 0,Y 452.391,Z 467.785,A -85,B 0,C 180,E1 -8174.38,E2 -8174.38} C_VEL
LIN {X 0,Y 452.453,Z 465.932,A -85,B 0,C 180,E1 -8175.609,E2 -8175.609} C_VEL
LIN {X 0,Y 452.56,Z 462.869,A -85,B 0,C 180,E1 -8176.987,E2 -8176.987} C_VEL
LIN {X 0,Y 452.741,Z 458.719,A -85,B 0,C 180,E1 -8178.357,E2 -8178.357} C_VEL
LIN {X 0,Y 452.949,Z 452.364,A -85,B 0,C 180,E1 -8179.947,E2 -8179.947} C_VEL
LIN {X 0,Y 453.323,Z 445.438,A -85,B 0,C 180,E1 -8181.306,E2 -8181.306} C_VEL
LIN {X 0,Y 453.787,Z 437.253,A -85,B 0,C 180,E1 -8182.595,E2 -8182.595} C_VEL
LIN {X 0,Y 454.178,Z 427.948,A -85,B 0,C 180,E1 -8183.781,E2 -8183.781} C_VEL
LIN {X 0,Y 454.733,Z 418.207,A -85,B 0,C 180,E1 -8184.79,E2 -8184.79} C_VEL
LIN {X 0,Y 455.31,Z 407.542,A -85,B 0,C 180,E1 -8185.684,E2 -8185.684} C_VEL
LIN {X 0,Y 455.844,Z 395.641,A -85,B 0,C 180,E1 -8186.464,E2 -8186.464} C_VEL
LIN {X 0,Y 456.239,Z 383.316,A -85,B 0,C 180,E1 -8187.075,E2 -8187.075} C_VEL
LIN {X 0,Y 456.569,Z 371.071,A -85,B 0,C 180,E1 -8187.505,E2 -8187.505} C_VEL
LIN {X 0,Y 456.818,Z 358.245,A -85,B 0,C 180,E1 -8187.779,E2 -8187.779} C_VEL
LIN {X 0,Y 457.421,Z 275.089,A -85,B 0,C 180,E1 -8189.092,E2 -8189.092} C_VEL
LIN {X 0,Y 454.664,Z 260,A -85,B 0,C 180,E1 -8189.435,E2 -8189.435} C_VEL
LIN {X 0,Y 454.411,Z 257.861,A -85,B 0,C 180,E1 -8189.556,E2 -8189.556} C_VEL
LIN {X 0,Y 455.163,Z 242.64,A -85,B 0,C 180,E1 -8192.655,E2 -8192.655} C_VEL
LIN {X 0,Y 455.156,Z 239.46,A -85,B 0,C 180,E1 -8193.319,E2 -8193.319} C_VEL
LIN {X 0,Y 453.68,Z 230.812,A -85,B 0,C 180,E1 -8195.221,E2 -8195.221} C_VEL
LIN {X 0,Y 453.656,Z 230.479,A -85,B 0,C 180,E1 -8195.556,E2 -8195.556} C_VEL
LIN {X 0,Y 453.609,Z 230.483,A -85,B 0,C 180,E1 -8198.015,E2 -8198.015} C_VEL
LIN {X 0,Y 453.57,Z 230.483,A -85,B 0,C 180,E1 -8201.62,E2 -8201.62} C_VEL
LIN {X 0,Y 453.517,Z 230.494,A -85,B 0,C 180,E1 -8204.356,E2 -8204.356} C_VEL
LIN {X 0,Y 453.486,Z 230.493,A -85,B 0,C 180,E1 -8207.125,E2 -8207.125} C_VEL
LIN {X 0,Y 453.49,Z 230.483,A -85,B 0,C 180,E1 -8209.934,E2 -8209.934} C_VEL
LIN {X 0,Y 453.479,Z 230.499,A -85,B 0,C 180,E1 -8212.795,E2 -8212.795} C_VEL
LIN {X 0,Y 453.486,Z 230.478,A -85,B 0,C 180,E1 -8216.005,E2 -8216.005} C_VEL
LIN {X 0,Y 453.483,Z 230.483,A -85,B 0,C 180,E1 -8218.713,E2 -8218.713} C_VEL
LIN {X 0,Y 453.492,Z 230.496,A -85,B 0,C 180,E1 -8221.797,E2 -8221.797} C_VEL
LIN {X 0,Y 453.466,Z 230.493,A -85,B 0,C 180,E1 -8224.99,E2 -8224.99} C_VEL
LIN {X 0,Y 453.465,Z 230.496,A -85,B 0,C 180,E1 -8228.311,E2 -8228.311} C_VEL
LIN {X 0,Y 453.479,Z 230.49,A -85,B 0,C 180,E1 -8230.61,E2 -8230.61} C_VEL
LIN {X 0,Y 453.507,Z 230.491,A -85,B 0,C 180,E1 -8234.215,E2 -8234.215} C_VEL
LIN {X 0,Y 453.481,Z 230.493,A -85,B 0,C 180,E1 -8237.015,E2 -8237.015} C_VEL
LIN {X 0,Y 453.506,Z 230.479,A -85,B 0,C 180,E1 -8240.559,E2 -8240.559} C_VEL
LIN {X 0,Y 453.431,Z 230.496,A -85,B 0,C 180,E1 -8243.922,E2 -8243.922} C_VEL
LIN {X 0,Y 453.457,Z 230.496,A -85,B 0,C 180,E1 -8247.156,E2 -8247.156} C_VEL
LIN {X 0,Y 453.49,Z 230.491,A -85,B 0,C 180,E1 -8250.276,E2 -8250.276} C_VEL
LIN {X 0,Y 453.493,Z 230.48,A -85,B 0,C 180,E1 -8253.299,E2 -8253.299} C_VEL
LIN {X 0,Y 453.486,Z 230.49,A -85,B 0,C 180,E1 -8256.243,E2 -8256.243} C_VEL
LIN {X 0,Y 453.491,Z 230.495,A -85,B 0,C 180,E1 -8259.123,E2 -8259.123} C_VEL
LIN {X 0,Y 453.497,Z 230.483,A -85,B 0,C 180,E1 -8261.949,E2 -8261.949} C_VEL
LIN {X 0,Y 453.527,Z 230.472,A -85,B 0,C 180,E1 -8264.731,E2 -8264.731} C_VEL
LIN {X 0,Y 453.591,Z 230.478,A -85,B 0,C 180,E1 -8267.477,E2 -8267.477} C_VEL
LIN {X 0,Y 453.586,Z 230.484,A -85,B 0,C 180,E1 -8271.091,E2 -8271.091} C_VEL
LIN {X 0,Y 453.673,Z 230.467,A -85,B 0,C 180,E1 -8273.779,E2 -8273.779} C_VEL
LIN {X 0,Y 453.739,Z 230.448,A -85,B 0,C 180,E1 -8277.341,E2 -8277.341} C_VEL
LIN {X 0,Y 453.819,Z 230.448,A -85,B 0,C 180,E1 -8280.004,E2 -8280.004} C_VEL
LIN {X 0,Y 453.742,Z 230.459,A -85,B 0,C 180,E1 -8282.667,E2 -8282.667} C_VEL
LIN {X 0,Y 453.652,Z 230.472,A -85,B 0,C 180,E1 -8286.229,E2 -8286.229} C_VEL
LIN {X 0,Y 453.591,Z 230.466,A -85,B 0,C 180,E1 -8288.917,E2 -8288.917} C_VEL
LIN {X 0,Y 453.566,Z 230.481,A -85,B 0,C 180,E1 -8292.532,E2 -8292.532} C_VEL
LIN {X 0,Y 453.548,Z 230.491,A -85,B 0,C 180,E1 -8296.199,E2 -8296.199} C_VEL
LIN {X 0,Y 453.521,Z 230.482,A -85,B 0,C 180,E1 -8299.042,E2 -8299.042} C_VEL
LIN {X 0,Y 453.482,Z 230.482,A -85,B 0,C 180,E1 -8301.839,E2 -8301.839} C_VEL
LIN {X 0,Y 453.505,Z 230.498,A -85,B 0,C 180,E1 -8304.738,E2 -8304.738} C_VEL
LIN {X 0,Y 453.535,Z 230.484,A -85,B 0,C 180,E1 -8307.961,E2 -8307.961} C_VEL
LIN {X 0,Y 453.47,Z 230.495,A -85,B 0,C 180,E1 -8311.527,E2 -8311.527} C_VEL
LIN {X 0,Y 453.489,Z 230.498,A -85,B 0,C 180,E1 -8314.778,E2 -8314.778} C_VEL
LIN {X 0,Y 453.466,Z 230.492,A -85,B 0,C 180,E1 -8318.314,E2 -8318.314} C_VEL
LIN {X 0,Y 453.502,Z 230.491,A -85,B 0,C 180,E1 -8320.611,E2 -8320.611} C_VEL
LIN {X 0,Y 453.468,Z 230.479,A -85,B 0,C 180,E1 -8324.224,E2 -8324.224} C_VEL
LIN {X 0,Y 453.456,Z 230.488,A -85,B 0,C 180,E1 -8327.005,E2 -8327.005} C_VEL
LIN {X 0,Y 453.503,Z 230.495,A -85,B 0,C 180,E1 -8329.411,E2 -8329.411} C_VEL
LIN {X 0,Y 453.457,Z 230.494,A -85,B 0,C 180,E1 -8332.811,E2 -8332.811} C_VEL
LIN {X 0,Y 453.485,Z 230.496,A -85,B 0,C 180,E1 -8336.089,E2 -8336.089} C_VEL
LIN {X 0,Y 453.485,Z 230.494,A -85,B 0,C 180,E1 -8339.242,E2 -8339.242} C_VEL
LIN {X 0,Y 453.541,Z 230.491,A -85,B 0,C 180,E1 -8342.298,E2 -8342.298} C_VEL
LIN {X 0,Y 453.542,Z 230.634,A -85,B 0,C 180,E1 -8344.839,E2 -8344.839} C_VEL
LIN {X 0,Y 455.566,Z 241.265,A -85,B 0,C 180,E1 -8347.075,E2 -8347.075} C_VEL
LIN {X 0,Y 455.155,Z 252.247,A -85,B 0,C 180,E1 -8349.198,E2 -8349.198} C_VEL
LIN {X 0,Y 454.485,Z 266.845,A -85,B 0,C 180,E1 -8351.985,E2 -8351.985} C_VEL
LIN {X 0,Y 454.409,Z 269.979,A -85,B 0,C 180,E1 -8352.531,E2 -8352.531} C_VEL
LIN {X 0,Y 457.444,Z 288.931,A -85,B 0,C 180,E1 -8352.971,E2 -8352.971} C_VEL
LIN {X 0,Y 456.704,Z 378.115,A -85,B 0,C 180,E1 -8354.406,E2 -8354.406} C_VEL
LIN {X 0,Y 456.33,Z 391.989,A -85,B 0,C 180,E1 -8354.822,E2 -8354.822} C_VEL
LIN {X 0,Y 455.863,Z 404.423,A -85,B 0,C 180,E1 -8355.378,E2 -8355.378} C_VEL
LIN {X 0,Y 455.342,Z 415.523,A -85,B 0,C 180,E1 -8356.045,E2 -8356.045} C_VEL
LIN {X 0,Y 454.808,Z 427.215,A -85,B 0,C 180,E1 -8356.949,E2 -8356.949} C_VEL
LIN {X 0,Y 454.286,Z 437.527,A -85,B 0,C 180,E1 -8357.945,E2 -8357.945} C_VEL
LIN {X 0,Y 453.736,Z 446.885,A -85,B 0,C 180,E1 -8359.063,E2 -8359.063} C_VEL
LIN {X 0,Y 453.261,Z 455.937,A -85,B 0,C 180,E1 -8360.405,E2 -8360.405} C_VEL
LIN {X 0,Y 452.948,Z 463.226,A -85,B 0,C 180,E1 -8361.749,E2 -8361.749} C_VEL
LIN {X 0,Y 452.728,Z 468.149,A -85,B 0,C 180,E1 -8362.866,E2 -8362.866} C_VEL
LIN {X 0,Y 452.593,Z 472.928,A -85,B 0,C 180,E1 -8364.207,E2 -8364.207} C_VEL
LIN {X 0,Y 452.491,Z 476.583,A -85,B 0,C 180,E1 -8365.546,E2 -8365.546} C_VEL
LIN {X 0,Y 452.458,Z 478.471,A -85,B 0,C 180,E1 -8366.438,E2 -8366.438} C_VEL
LIN {X 0,Y 452.494,Z 479.899,A -85,B 0,C 180,E1 -8367.33,E2 -8367.33} C_VEL
LIN {X 0,Y 452.406,Z 481.534,A -85,B 0,C 180,E1 -8369.11,E2 -8369.11} C_VEL
LIN {X 0,Y 452.41,Z 481.773,A -85,B 0,C 180,E1 -8370,E2 -8370} C_VEL
LIN {X 0,Y 452.406,Z 481.585,A -85,B 0,C 180,E1 -8370.89,E2 -8370.89} C_VEL
LIN {X 0,Y 452.494,Z 480.018,A -85,B 0,C 180,E1 -8372.671,E2 -8372.671} C_VEL
LIN {X 0,Y 452.459,Z 478.647,A -85,B 0,C 180,E1 -8373.562,E2 -8373.562} C_VEL
LIN {X 0,Y 452.558,Z 475.75,A -85,B 0,C 180,E1 -8374.9,E2 -8374.9} C_VEL
LIN {X 0,Y 452.638,Z 471.241,A -85,B 0,C 180,E1 -8376.416,E2 -8376.416} C_VEL
LIN {X 0,Y 452.909,Z 464.798,A -85,B 0,C 180,E1 -8378.028,E2 -8378.028} C_VEL
LIN {X 0,Y 453.24,Z 457.976,A -85,B 0,C 180,E1 -8379.371,E2 -8379.371} C_VEL
LIN {X 0,Y 453.686,Z 449.477,A -85,B 0,C 180,E1 -8380.713,E2 -8380.713} C_VEL
LIN {X 0,Y 454.288,Z 440.746,A -85,B 0,C 180,E1 -8381.829,E2 -8381.829} C_VEL
LIN {X 0,Y 454.881,Z 429.928,A -85,B 0,C 180,E1 -8382.954,E2 -8382.954} C_VEL
LIN {X 0,Y 455.4,Z 419.299,A -85,B 0,C 180,E1 -8383.84,E2 -8383.84} C_VEL
LIN {X 0,Y 456.027,Z 407.287,A -85,B 0,C 180,E1 -8384.618,E2 -8384.618} C_VEL
LIN {X 0,Y 456.572,Z 394.777,A -85,B 0,C 180,E1 -8385.227,E2 -8385.227} C_VEL
LIN {X 0,Y 456.959,Z 382.721,A -85,B 0,C 180,E1 -8385.642,E2 -8385.642} C_VEL
LIN {X 0,Y 457.215,Z 369.393,A -85,B 0,C 180,E1 -8385.919,E2 -8385.919} C_VEL
LIN {X 0,Y 457.869,Z 288.876,A -85,B 0,C 180,E1 -8387.21,E2 -8387.21} C_VEL
LIN {X 0,Y 454.608,Z 270.2,A -85,B 0,C 180,E1 -8387.676,E2 -8387.676} C_VEL
LIN {X 0,Y 454.58,Z 269.028,A -85,B 0,C 180,E1 -8387.802,E2 -8387.802} C_VEL
LIN {X 0,Y 455.439,Z 250.977,A -85,B 0,C 180,E1 -8391.262,E2 -8391.262} C_VEL
LIN {X 0,Y 455.828,Z 242.534,A -85,B 0,C 180,E1 -8392.912,E2 -8392.912} C_VEL
LIN {X 0,Y 453.742,Z 231.733,A -85,B 0,C 180,E1 -8395.211,E2 -8395.211} C_VEL
LIN {X 0,Y 453.524,Z 230.519,A -85,B 0,C 180,E1 -8395.562,E2 -8395.562} C_VEL
LIN {X 0,Y 453.517,Z 230.491,A -85,B 0,C 180,E1 -8398.711,E2 -8398.711} C_VEL
LIN {X 0,Y 453.475,Z 230.5,A -85,B 0,C 180,E1 -8401.799,E2 -8401.799} C_VEL
LIN {X 0,Y 453.49,Z 230.492,A -85,B 0,C 180,E1 -8404.989,E2 -8404.989} C_VEL
LIN {X 0,Y 453.468,Z 230.495,A -85,B 0,C 180,E1 -8408.311,E2 -8408.311} C_VEL
LIN {X 0,Y 453.482,Z 230.498,A -85,B 0,C 180,E1 -8410.61,E2 -8410.61} C_VEL
LIN {X 0,Y 453.471,Z 230.497,A -85,B 0,C 180,E1 -8414.221,E2 -8414.221} C_VEL
LIN {X 0,Y 453.459,Z 230.488,A -85,B 0,C 180,E1 -8417.002,E2 -8417.002} C_VEL
LIN {X 0,Y 453.505,Z 230.491,A -85,B 0,C 180,E1 -8419.408,E2 -8419.408} C_VEL
LIN {X 0,Y 453.46,Z 230.504,A -85,B 0,C 180,E1 -8422.808,E2 -8422.808} C_VEL
LIN {X 0,Y 453.477,Z 230.495,A -85,B 0,C 180,E1 -8426.084,E2 -8426.084} C_VEL
LIN {X 0,Y 453.484,Z 230.498,A -85,B 0,C 180,E1 -8429.238,E2 -8429.238} C_VEL
LIN {X 0,Y 453.484,Z 230.49,A -85,B 0,C 180,E1 -8432.291,E2 -8432.291} C_VEL
LIN {X 0,Y 453.479,Z 230.495,A -85,B 0,C 180,E1 -8435.26,E2 -8435.26} C_VEL
LIN {X 0,Y 453.489,Z 230.492,A -85,B 0,C 180,E1 -8438.412,E2 -8438.412} C_VEL
LIN {X 0,Y 453.531,Z 230.486,A -85,B 0,C 180,E1 -8441.006,E2 -8441.006} C_VEL
LIN {X 0,Y 453.577,Z 230.478,A -85,B 0,C 180,E1 -8443.877,E2 -8443.877} C_VEL
LIN {X 0,Y 453.571,Z 230.489,A -85,B 0,C 180,E1 -8447.468,E2 -8447.468} C_VEL
LIN {X 0,Y 453.584,Z 230.481,A -85,B 0,C 180,E1 -8451.083,E2 -8451.083} C_VEL
LIN {X 0,Y 453.66,Z 230.472,A -85,B 0,C 180,E1 -8453.771,E2 -8453.771} C_VEL
LIN {X 0,Y 453.732,Z 230.463,A -85,B 0,C 180,E1 -8457.333,E2 -8457.333} C_VEL
LIN {X 0,Y 453.82,Z 230.455,A -85,B 0,C 180,E1 -8459.996,E2 -8459.996} C_VEL
LIN {X 0,Y 453.734,Z 230.458,A -85,B 0,C 180,E1 -8462.659,E2 -8462.659} C_VEL
LIN {X 0,Y 453.648,Z 230.477,A -85,B 0,C 180,E1 -8466.221,E2 -8466.221} C_VEL
LIN {X 0,Y 453.581,Z 230.483,A -85,B 0,C 180,E1 -8468.909,E2 -8468.909} C_VEL
LIN {X 0,Y 453.557,Z 230.488,A -85,B 0,C 180,E1 -8472.524,E2 -8472.524} C_VEL
LIN {X 0,Y 453.535,Z 230.487,A -85,B 0,C 180,E1 -8476.191,E2 -8476.191} C_VEL
LIN {X 0,Y 453.506,Z 230.494,A -85,B 0,C 180,E1 -8479.035,E2 -8479.035} C_VEL
LIN {X 0,Y 453.464,Z 230.493,A -85,B 0,C 180,E1 -8481.831,E2 -8481.831} C_VEL
LIN {X 0,Y 453.498,Z 230.495,A -85,B 0,C 180,E1 -8484.73,E2 -8484.73} C_VEL
LIN {X 0,Y 453.519,Z 230.488,A -85,B 0,C 180,E1 -8487.956,E2 -8487.956} C_VEL
LIN {X 0,Y 453.444,Z 230.498,A -85,B 0,C 180,E1 -8491.52,E2 -8491.52} C_VEL
LIN {X 0,Y 453.465,Z 230.496,A -85,B 0,C 180,E1 -8494.773,E2 -8494.773} C_VEL
LIN {X 0,Y 453.46,Z 230.493,A -85,B 0,C 180,E1 -8498.305,E2 -8498.305} C_VEL
LIN {X 0,Y 453.488,Z 230.493,A -85,B 0,C 180,E1 -8500.602,E2 -8500.602} C_VEL
LIN {X 0,Y 453.451,Z 230.5,A -85,B 0,C 180,E1 -8503.243,E2 -8503.243} C_VEL
LIN {X 0,Y 453.444,Z 230.506,A -85,B 0,C 180,E1 -8505.776,E2 -8505.776} C_VEL
LIN {X 0,Y 453.51,Z 230.601,A -85,B 0,C 180,E1 -8508.68,E2 -8508.68} C_VEL
LIN {X 0,Y 455.144,Z 238.878,A -85,B 0,C 180,E1 -8510.53,E2 -8510.53} C_VEL
LIN {X 0,Y 455.216,Z 243.99,A -85,B 0,C 180,E1 -8511.581,E2 -8511.581} C_VEL
LIN {X 0,Y 454.669,Z 257.753,A -85,B 0,C 180,E1 -8514.301,E2 -8514.301} C_VEL
LIN {X 0,Y 454.95,Z 259.698,A -85,B 0,C 180,E1 -8514.418,E2 -8514.418} C_VEL
LIN {X 0,Y 457.991,Z 275.87,A -85,B 0,C 180,E1 -8514.821,E2 -8514.821} C_VEL
LIN {X 0,Y 457.077,Z 366.001,A -85,B 0,C 180,E1 -8516.284,E2 -8516.284} C_VEL
LIN {X 0,Y 456.703,Z 379.875,A -85,B 0,C 180,E1 -8516.706,E2 -8516.706} C_VEL
LIN {X 0,Y 456.269,Z 391.868,A -85,B 0,C 180,E1 -8517.246,E2 -8517.246} C_VEL
LIN {X 0,Y 455.748,Z 404.156,A -85,B 0,C 180,E1 -8517.999,E2 -8517.999} C_VEL
LIN {X 0,Y 455.198,Z 415.042,A -85,B 0,C 180,E1 -8518.854,E2 -8518.854} C_VEL
LIN {X 0,Y 454.586,Z 425.601,A -85,B 0,C 180,E1 -8519.887,E2 -8519.887} C_VEL
LIN {X 0,Y 454.009,Z 435.265,A -85,B 0,C 180,E1 -8521.069,E2 -8521.069} C_VEL
LIN {X 0,Y 453.533,Z 443.424,A -85,B 0,C 180,E1 -8522.297,E2 -8522.297} C_VEL
LIN {X 0,Y 453.376,Z 446.019,A -85,B 0,C 180,E1 -8522.745,E2 -8522.745} C_VEL
LIN {X 0,Y 452.525,Z 449.364,A -85,B 0,C 180,E1 -8523.357,E2 -8523.357} C_VEL
LIN {X 0,Y 449.39,Z 454.362,A -85,B 0,C 180,E1 -8524.374,E2 -8524.374} C_VEL
LIN {X 0,Y 446.328,Z 458.665,A -85,B 0,C 180,E1 -8525.448,E2 -8525.448} C_VEL
LIN {X 0,Y 445.597,Z 460.924,A -85,B 0,C 180,E1 -8526.141,E2 -8526.141} C_VEL
LIN {X 0,Y 445.401,Z 464.992,A -85,B 0,C 180,E1 -8527.747,E2 -8527.747} C_VEL
LIN {X 0,Y 445.334,Z 466.76,A -85,B 0,C 180,E1 -8528.717,E2 -8528.717} C_VEL
LIN {X 0,Y 445.266,Z 468.075,A -85,B 0,C 180,E1 -8529.681,E2 -8529.681} C_VEL
LIN {X 0,Y 445.257,Z 469.221,A -85,B 0,C 180,E1 -8531.251,E2 -8531.251} C_VEL
LIN {X 0,Y 445.201,Z 469.247,A -85,B 0,C 180,E1 -8532.546,E2 -8532.546} C_VEL
LIN {X 0,Y 445.292,Z 468.017,A -85,B 0,C 180,E1 -8534.289,E2 -8534.289} C_VEL
LIN {X 0,Y 445.348,Z 466.485,A -85,B 0,C 180,E1 -8535.375,E2 -8535.375} C_VEL
LIN {X 0,Y 445.45,Z 463.618,A -85,B 0,C 180,E1 -8536.775,E2 -8536.775} C_VEL
LIN {X 0,Y 445.628,Z 459.688,A -85,B 0,C 180,E1 -8538.169,E2 -8538.169} C_VEL
LIN {X 0,Y 445.828,Z 454.607,A -85,B 0,C 180,E1 -8539.555,E2 -8539.555} C_VEL
LIN {X 0,Y 446.121,Z 448.22,A -85,B 0,C 180,E1 -8540.936,E2 -8540.936} C_VEL
LIN {X 0,Y 446.541,Z 440.791,A -85,B 0,C 180,E1 -8542.223,E2 -8542.223} C_VEL
LIN {X 0,Y 447.022,Z 432.056,A -85,B 0,C 180,E1 -8543.455,E2 -8543.455} C_VEL
LIN {X 0,Y 447.581,Z 422.122,A -85,B 0,C 180,E1 -8544.594,E2 -8544.594} C_VEL
LIN {X 0,Y 448.094,Z 412.359,A -85,B 0,C 180,E1 -8545.502,E2 -8545.502} C_VEL
LIN {X 0,Y 448.632,Z 401.766,A -85,B 0,C 180,E1 -8546.295,E2 -8546.295} C_VEL
LIN {X 0,Y 449.199,Z 389.001,A -85,B 0,C 180,E1 -8547.029,E2 -8547.029} C_VEL
LIN {X 0,Y 449.59,Z 376.392,A -85,B 0,C 180,E1 -8547.558,E2 -8547.558} C_VEL
LIN {X 0,Y 449.91,Z 363.452,A -85,B 0,C 180,E1 -8547.907,E2 -8547.907} C_VEL
LIN {X 0,Y 450.623,Z 276.077,A -85,B 0,C 180,E1 -8549.316,E2 -8549.316} C_VEL
LIN {X 0,Y 447.478,Z 258.484,A -85,B 0,C 180,E1 -8549.747,E2 -8549.747} C_VEL
LIN {X 0,Y 447.597,Z 254.747,A -85,B 0,C 180,E1 -8550.45,E2 -8550.45} C_VEL
LIN {X 0,Y 448.282,Z 241.812,A -85,B 0,C 180,E1 -8553.145,E2 -8553.145} C_VEL
LIN {X 0,Y 446.626,Z 231.409,A -85,B 0,C 180,E1 -8555.502,E2 -8555.502} C_VEL
LIN {X 0,Y 446.558,Z 231.363,A -85,B 0,C 180,E1 -8558.143,E2 -8558.143} C_VEL
LIN {X 0,Y 446.494,Z 231.369,A -85,B 0,C 180,E1 -8560.887,E2 -8560.887} C_VEL
LIN {X 0,Y 446.474,Z 231.367,A -85,B 0,C 180,E1 -8563.657,E2 -8563.657} C_VEL
LIN {X 0,Y 446.452,Z 231.373,A -85,B 0,C 180,E1 -8566.46,E2 -8566.46} C_VEL
LIN {X 0,Y 446.429,Z 231.364,A -85,B 0,C 180,E1 -8569.305,E2 -8569.305} C_VEL
LIN {X 0,Y 446.422,Z 231.373,A -85,B 0,C 180,E1 -8572.199,E2 -8572.199} C_VEL
LIN {X 0,Y 446.431,Z 231.365,A -85,B 0,C 180,E1 -8575.153,E2 -8575.153} C_VEL
LIN {X 0,Y 446.477,Z 231.354,A -85,B 0,C 180,E1 -8578.19,E2 -8578.19} C_VEL
LIN {X 0,Y 446.448,Z 231.373,A -85,B 0,C 180,E1 -8581.793,E2 -8581.793} C_VEL
LIN {X 0,Y 446.415,Z 231.372,A -85,B 0,C 180,E1 -8585.061,E2 -8585.061} C_VEL
LIN {X 0,Y 446.415,Z 231.376,A -85,B 0,C 180,E1 -8588.089,E2 -8588.089} C_VEL
LIN {X 0,Y 446.411,Z 231.37,A -85,B 0,C 180,E1 -8590.924,E2 -8590.924} C_VEL
LIN {X 0,Y 446.457,Z 231.367,A -85,B 0,C 180,E1 -8593.838,E2 -8593.838} C_VEL
LIN {X 0,Y 446.458,Z 231.37,A -85,B 0,C 180,E1 -8596.395,E2 -8596.395} C_VEL
LIN {X 0,Y 446.439,Z 231.371,A -85,B 0,C 180,E1 -8599.809,E2 -8599.809} C_VEL
LIN {X 0,Y 446.406,Z 231.366,A -85,B 0,C 180,E1 -8602.128,E2 -8602.128} C_VEL
LIN {X 0,Y 446.404,Z 231.373,A -85,B 0,C 180,E1 -8605.482,E2 -8605.482} C_VEL
LIN {X 0,Y 446.406,Z 231.374,A -85,B 0,C 180,E1 -8608.705,E2 -8608.705} C_VEL
LIN {X 0,Y 446.462,Z 231.352,A -85,B 0,C 180,E1 -8611.826,E2 -8611.826} C_VEL
LIN {X 0,Y 446.44,Z 231.37,A -85,B 0,C 180,E1 -8614.852,E2 -8614.852} C_VEL
LIN {X 0,Y 446.452,Z 231.37,A -85,B 0,C 180,E1 -8618.242,E2 -8618.242} C_VEL
LIN {X 0,Y 446.442,Z 231.363,A -85,B 0,C 180,E1 -8621.654,E2 -8621.654} C_VEL
LIN {X 0,Y 446.495,Z 231.346,A -85,B 0,C 180,E1 -8624.484,E2 -8624.484} C_VEL
LIN {X 0,Y 446.53,Z 231.353,A -85,B 0,C 180,E1 -8628.198,E2 -8628.198} C_VEL
LIN {X 0,Y 446.593,Z 231.352,A -85,B 0,C 180,E1 -8631.862,E2 -8631.862} C_VEL
LIN {X 0,Y 446.641,Z 231.339,A -85,B 0,C 180,E1 -8634.587,E2 -8634.587} C_VEL
LIN {X 0,Y 446.66,Z 231.326,A -85,B 0,C 180,E1 -8638.201,E2 -8638.201} C_VEL
LIN {X 0,Y 446.789,Z 231.323,A -85,B 0,C 180,E1 -8640.004,E2 -8640.004} C_VEL
LIN {X 0,Y 446.689,Z 231.337,A -85,B 0,C 180,E1 -8642.709,E2 -8642.709} C_VEL
LIN {X 0,Y 446.62,Z 231.346,A -85,B 0,C 180,E1 -8646.328,E2 -8646.328} C_VEL
LIN {X 0,Y 446.537,Z 231.344,A -85,B 0,C 180,E1 -8649.059,E2 -8649.059} C_VEL
LIN {X 0,Y 446.524,Z 231.357,A -85,B 0,C 180,E1 -8652.733,E2 -8652.733} C_VEL
LIN {X 0,Y 446.499,Z 231.37,A -85,B 0,C 180,E1 -8656.231,E2 -8656.231} C_VEL
LIN {X 0,Y 446.473,Z 231.358,A -85,B 0,C 180,E1 -8659.306,E2 -8659.306} C_VEL
LIN {X 0,Y 446.423,Z 231.364,A -85,B 0,C 180,E1 -8662.203,E2 -8662.203} C_VEL
LIN {X 0,Y 446.447,Z 231.372,A -85,B 0,C 180,E1 -8665.156,E2 -8665.156} C_VEL
LIN {X 0,Y 446.492,Z 231.363,A -85,B 0,C 180,E1 -8668.181,E2 -8668.181} C_VEL
LIN {X 0,Y 446.422,Z 231.371,A -85,B 0,C 180,E1 -8671.776,E2 -8671.776} C_VEL
LIN {X 0,Y 446.429,Z 231.375,A -85,B 0,C 180,E1 -8674.526,E2 -8674.526} C_VEL
LIN {X 0,Y 446.418,Z 231.369,A -85,B 0,C 180,E1 -8678.081,E2 -8678.081} C_VEL
LIN {X 0,Y 446.427,Z 231.375,A -85,B 0,C 180,E1 -8681.394,E2 -8681.394} C_VEL
LIN {X 0,Y 446.458,Z 231.352,A -85,B 0,C 180,E1 -8685.106,E2 -8685.106} C_VEL
LIN {X 0,Y 446.427,Z 231.371,A -85,B 0,C 180,E1 -8688.609,E2 -8688.609} C_VEL
LIN {X 0,Y 446.419,Z 231.373,A -85,B 0,C 180,E1 -8691.923,E2 -8691.923} C_VEL
LIN {X 0,Y 446.437,Z 231.374,A -85,B 0,C 180,E1 -8695.478,E2 -8695.478} C_VEL
LIN {X 0,Y 446.424,Z 231.374,A -85,B 0,C 180,E1 -8698.701,E2 -8698.701} C_VEL
LIN {X 0,Y 446.495,Z 231.371,A -85,B 0,C 180,E1 -8701.823,E2 -8701.823} C_VEL
LIN {X 0,Y 446.495,Z 231.543,A -85,B 0,C 180,E1 -8704.663,E2 -8704.663} C_VEL
LIN {X 0,Y 448.54,Z 242.231,A -85,B 0,C 180,E1 -8706.939,E2 -8706.939} C_VEL
LIN {X 0,Y 448.439,Z 248.343,A -85,B 0,C 180,E1 -8708.148,E2 -8708.148} C_VEL
LIN {X 0,Y 447.683,Z 264.186,A -85,B 0,C 180,E1 -8711.227,E2 -8711.227} C_VEL
LIN {X 0,Y 447.409,Z 269.751,A -85,B 0,C 180,E1 -8712.264,E2 -8712.264} C_VEL
LIN {X 0,Y 448.311,Z 275.598,A -85,B 0,C 180,E1 -8712.43,E2 -8712.43} C_VEL
LIN {X 0,Y 450.661,Z 290.823,A -85,B 0,C 180,E1 -8712.765,E2 -8712.765} C_VEL
LIN {X 0,Y 449.882,Z 377.093,A -85,B 0,C 180,E1 -8714.164,E2 -8714.164} C_VEL
LIN {X 0,Y 449.462,Z 390.526,A -85,B 0,C 180,E1 -8714.556,E2 -8714.556} C_VEL
LIN {X 0,Y 449.025,Z 402.776,A -85,B 0,C 180,E1 -8715.092,E2 -8715.092} C_VEL
LIN {X 0,Y 448.405,Z 415.113,A -85,B 0,C 180,E1 -8715.825,E2 -8715.825} C_VEL
LIN {X 0,Y 447.857,Z 426.864,A -85,B 0,C 180,E1 -8716.743,E2 -8716.743} C_VEL
LIN {X 0,Y 447.334,Z 437.221,A -85,B 0,C 180,E1 -8717.755,E2 -8717.755} C_VEL
LIN {X 0,Y 446.733,Z 446.628,A -85,B 0,C 180,E1 -8718.889,E2 -8718.889} C_VEL
LIN {X 0,Y 446.235,Z 455.707,A -85,B 0,C 180,E1 -8720.253,E2 -8720.253} C_VEL
LIN {X 0,Y 445.884,Z 463.02,A -85,B 0,C 180,E1 -8721.617,E2 -8721.617} C_VEL
LIN {X 0,Y 445.65,Z 467.963,A -85,B 0,C 180,E1 -8722.752,E2 -8722.752} C_VEL
LIN {X 0,Y 445.504,Z 472.165,A -85,B 0,C 180,E1 -8723.926,E2 -8723.926} C_VEL
LIN {X 0,Y 445.418,Z 476.434,A -85,B 0,C 180,E1 -8725.475,E2 -8725.475} C_VEL
LIN {X 0,Y 445.358,Z 478.331,A -85,B 0,C 180,E1 -8726.381,E2 -8726.381} C_VEL
LIN {X 0,Y 445.401,Z 479.775,A -85,B 0,C 180,E1 -8727.287,E2 -8727.287} C_VEL
LIN {X 0,Y 445.318,Z 481.425,A -85,B 0,C 180,E1 -8729.096,E2 -8729.096} C_VEL
LIN {X 0,Y 445.32,Z 481.671,A -85,B 0,C 180,E1 -8730,E2 -8730} C_VEL
LIN {X 0,Y 445.319,Z 481.497,A -85,B 0,C 180,E1 -8730.905,E2 -8730.905} C_VEL
LIN {X 0,Y 445.402,Z 479.944,A -85,B 0,C 180,E1 -8732.714,E2 -8732.714} C_VEL
LIN {X 0,Y 445.359,Z 478.58,A -85,B 0,C 180,E1 -8733.619,E2 -8733.619} C_VEL
LIN {X 0,Y 445.491,Z 475.699,A -85,B 0,C 180,E1 -8734.978,E2 -8734.978} C_VEL
LIN {X 0,Y 445.613,Z 470.395,A -85,B 0,C 180,E1 -8736.748,E2 -8736.748} C_VEL
LIN {X 0,Y 445.93,Z 463.777,A -85,B 0,C 180,E1 -8738.383,E2 -8738.383} C_VEL
LIN {X 0,Y 446.301,Z 456.706,A -85,B 0,C 180,E1 -8739.746,E2 -8739.746} C_VEL
LIN {X 0,Y 446.833,Z 447.895,A -85,B 0,C 180,E1 -8741.109,E2 -8741.109} C_VEL
LIN {X 0,Y 447.485,Z 437.9,A -85,B 0,C 180,E1 -8742.356,E2 -8742.356} C_VEL
LIN {X 0,Y 447.984,Z 428.69,A -85,B 0,C 180,E1 -8743.29,E2 -8743.29} C_VEL
LIN {X 0,Y 448.614,Z 417.969,A -85,B 0,C 180,E1 -8744.169,E2 -8744.169} C_VEL
LIN {X 0,Y 449.262,Z 405.659,A -85,B 0,C 180,E1 -8744.959,E2 -8744.959} C_VEL
LIN {X 0,Y 449.805,Z 393.995,A -85,B 0,C 180,E1 -8745.52,E2 -8745.52} C_VEL
LIN {X 0,Y 450.203,Z 381.505,A -85,B 0,C 180,E1 -8745.941,E2 -8745.941} C_VEL
LIN {X 0,Y 450.508,Z 365.711,A -85,B 0,C 180,E1 -8746.25,E2 -8746.25} C_VEL
LIN {X 0,Y 451.09,Z 289.398,A -85,B 0,C 180,E1 -8747.495,E2 -8747.495} C_VEL
LIN {X 0,Y 447.675,Z 269.735,A -85,B 0,C 180,E1 -8748.006,E2 -8748.006} C_VEL
LIN {X 0,Y 448.119,Z 259.783,A -85,B 0,C 180,E1 -8749.888,E2 -8749.888} C_VEL
LIN {X 0,Y 448.935,Z 245.498,A -85,B 0,C 180,E1 -8752.702,E2 -8752.702} C_VEL
LIN {X 0,Y 448.26,Z 240.22,A -85,B 0,C 180,E1 -8753.811,E2 -8753.811} C_VEL
LIN {X 0,Y 446.482,Z 231.471,A -85,B 0,C 180,E1 -8755.775,E2 -8755.775} C_VEL
LIN {X 0,Y 446.498,Z 231.37,A -85,B 0,C 180,E1 -8758.178,E2 -8758.178} C_VEL
LIN {X 0,Y 446.43,Z 231.377,A -85,B 0,C 180,E1 -8761.774,E2 -8761.774} C_VEL
LIN {X 0,Y 446.44,Z 231.373,A -85,B 0,C 180,E1 -8764.522,E2 -8764.522} C_VEL
LIN {X 0,Y 446.421,Z 231.375,A -85,B 0,C 180,E1 -8768.077,E2 -8768.077} C_VEL
LIN {X 0,Y 446.422,Z 231.373,A -85,B 0,C 180,E1 -8771.392,E2 -8771.392} C_VEL
LIN {X 0,Y 446.433,Z 231.374,A -85,B 0,C 180,E1 -8774.891,E2 -8774.891} C_VEL
LIN {X 0,Y 446.433,Z 231.361,A -85,B 0,C 180,E1 -8777.723,E2 -8777.723} C_VEL
LIN {X 0,Y 446.42,Z 231.375,A -85,B 0,C 180,E1 -8780.967,E2 -8780.967} C_VEL
LIN {X 0,Y 446.426,Z 231.375,A -85,B 0,C 180,E1 -8784.372,E2 -8784.372} C_VEL
LIN {X 0,Y 446.427,Z 231.369,A -85,B 0,C 180,E1 -8787.636,E2 -8787.636} C_VEL
LIN {X 0,Y 446.432,Z 231.377,A -85,B 0,C 180,E1 -8790.786,E2 -8790.786} C_VEL
LIN {X 0,Y 446.445,Z 231.37,A -85,B 0,C 180,E1 -8793.843,E2 -8793.843} C_VEL
LIN {X 0,Y 446.432,Z 231.371,A -85,B 0,C 180,E1 -8796.82,E2 -8796.82} C_VEL
LIN {X 0,Y 446.452,Z 231.367,A -85,B 0,C 180,E1 -8799.734,E2 -8799.734} C_VEL
LIN {X 0,Y 446.464,Z 231.368,A -85,B 0,C 180,E1 -8802.594,E2 -8802.594} C_VEL
LIN {X 0,Y 446.475,Z 231.366,A -85,B 0,C 180,E1 -8805.409,E2 -8805.409} C_VEL
LIN {X 0,Y 446.523,Z 231.358,A -85,B 0,C 180,E1 -8808.19,E2 -8808.19} C_VEL
LIN {X 0,Y 446.532,Z 231.359,A -85,B 0,C 180,E1 -8810.941,E2 -8810.941} C_VEL
LIN {X 0,Y 446.63,Z 231.348,A -85,B 0,C 180,E1 -8813.672,E2 -8813.672} C_VEL
LIN {X 0,Y 446.679,Z 231.341,A -85,B 0,C 180,E1 -8817.291,E2 -8817.291} C_VEL
LIN {X 0,Y 446.79,Z 231.331,A -85,B 0,C 180,E1 -8819.996,E2 -8819.996} C_VEL
LIN {X 0,Y 446.681,Z 231.336,A -85,B 0,C 180,E1 -8822.701,E2 -8822.701} C_VEL
LIN {X 0,Y 446.616,Z 231.351,A -85,B 0,C 180,E1 -8826.32,E2 -8826.32} C_VEL
LIN {X 0,Y 446.515,Z 231.364,A -85,B 0,C 180,E1 -8829.966,E2 -8829.966} C_VEL
LIN {X 0,Y 446.515,Z 231.367,A -85,B 0,C 180,E1 -8832.725,E2 -8832.725} C_VEL
LIN {X 0,Y 446.486,Z 231.365,A -85,B 0,C 180,E1 -8836.223,E2 -8836.223} C_VEL
LIN {X 0,Y 446.457,Z 231.37,A -85,B 0,C 180,E1 -8839.299,E2 -8839.299} C_VEL
LIN {X 0,Y 446.405,Z 231.373,A -85,B 0,C 180,E1 -8842.195,E2 -8842.195} C_VEL
LIN {X 0,Y 446.441,Z 231.366,A -85,B 0,C 180,E1 -8845.148,E2 -8845.148} C_VEL
LIN {X 0,Y 446.466,Z 231.367,A -85,B 0,C 180,E1 -8848.174,E2 -8848.174} C_VEL
LIN {X 0,Y 446.397,Z 231.377,A -85,B 0,C 180,E1 -8851.77,E2 -8851.77} C_VEL
LIN {X 0,Y 446.406,Z 231.374,A -85,B 0,C 180,E1 -8854.518,E2 -8854.518} C_VEL
LIN {X 0,Y 446.413,Z 231.371,A -85,B 0,C 180,E1 -8858.079,E2 -8858.079} C_VEL
LIN {X 0,Y 446.419,Z 231.374,A -85,B 0,C 180,E1 -8860.916,E2 -8860.916} C_VEL
LIN {X 0,Y 446.414,Z 231.38,A -85,B 0,C 180,E1 -8863.836,E2 -8863.836} C_VEL
LIN {X 0,Y 446.414,Z 231.377,A -85,B 0,C 180,E1 -8866.393,E2 -8866.393} C_VEL
LIN {X 0,Y 446.494,Z 231.584,A -85,B 0,C 180,E1 -8868.467,E2 -8868.467} C_VEL
LIN {X 0,Y 448.33,Z 241.036,A -85,B 0,C 180,E1 -8870.589,E2 -8870.589} C_VEL
LIN {X 0,Y 448.104,Z 249.333,A -85,B 0,C 180,E1 -8872.289,E2 -8872.289} C_VEL
LIN {X 0,Y 447.761,Z 258.092,A -85,B 0,C 180,E1 -8874.022,E2 -8874.022} C_VEL
LIN {X 0,Y 448.872,Z 263.62,A -85,B 0,C 180,E1 -8874.208,E2 -8874.208} C_VEL
LIN {X 0,Y 451.268,Z 276.492,A -85,B 0,C 180,E1 -8874.535,E2 -8874.535} C_VEL
LIN {X 0,Y 450.313,Z 366.303,A -85,B 0,C 180,E1 -8876.019,E2 -8876.019} C_VEL
LIN {X 0,Y 449.963,Z 379.548,A -85,B 0,C 180,E1 -8876.426,E2 -8876.426} C_VEL
LIN {X 0,Y 449.442,Z 392.432,A -85,B 0,C 180,E1 -8877.013,E2 -8877.013} C_VEL
LIN {X 0,Y 448.913,Z 403.576,A -85,B 0,C 180,E1 -8877.703,E2 -8877.703} C_VEL
LIN {X 0,Y 448.357,Z 414.742,A -85,B 0,C 180,E1 -8878.587,E2 -8878.587} C_VEL
LIN {X 0,Y 447.718,Z 424.623,A -85,B 0,C 180,E1 -8879.556,E2 -8879.556} C_VEL
LIN {X 0,Y 447.166,Z 433.224,A -85,B 0,C 180,E1 -8880.584,E2 -8880.584} C_VEL
LIN {X 0,Y 446.624,Z 441.798,A -85,B 0,C 180,E1 -8881.831,E2 -8881.831} C_VEL
LIN {X 0,Y 446.101,Z 449.966,A -85,B 0,C 180,E1 -8883.32,E2 -8883.32} C_VEL
LIN {X 0,Y 445.793,Z 456.409,A -85,B 0,C 180,E1 -8884.807,E2 -8884.807} C_VEL
LIN {X 0,Y 445.597,Z 460.924,A -85,B 0,C 180,E1 -8886.141,E2 -8886.141} C_VEL
LIN {X 0,Y 444.873,Z 462.968,A -85,B 0,C 180,E1 -8886.847,E2 -8886.847} C_VEL
LIN {X 0,Y 441.871,Z 465.66,A -85,B 0,C 180,E1 -8888.017,E2 -8888.017} C_VEL
LIN {X 0,Y 439.341,Z 467.354,A -85,B 0,C 180,E1 -8888.98,E2 -8888.98} C_VEL
LIN {X 0,Y 438.18,Z 468.419,A -85,B 0,C 180,E1 -8889.862,E2 -8889.862} C_VEL
LIN {X 0,Y 438.153,Z 468.485,A -85,B 0,C 180,E1 -8889.99,E2 -8889.99} C_VEL
LIN {X 0,Y 438.173,Z 469.337,A -85,B 0,C 180,E1 -8891.289,E2 -8891.289} C_VEL
LIN {X 0,Y 438.127,Z 469.394,A -85,B 0,C 180,E1 -8892.255,E2 -8892.255} C_VEL
LIN {X 0,Y 438.138,Z 469.039,A -85,B 0,C 180,E1 -8893.218,E2 -8893.218} C_VEL
LIN {X 0,Y 438.197,Z 468.247,A -85,B 0,C 180,E1 -8894.194,E2 -8894.194} C_VEL
LIN {X 0,Y 438.254,Z 467.016,A -85,B 0,C 180,E1 -8895.132,E2 -8895.132} C_VEL
LIN {X 0,Y 438.328,Z 464.349,A -85,B 0,C 180,E1 -8896.556,E2 -8896.556} C_VEL
LIN {X 0,Y 438.496,Z 460.627,A -85,B 0,C 180,E1 -8897.974,E2 -8897.974} C_VEL
LIN {X 0,Y 438.727,Z 455.76,A -85,B 0,C 180,E1 -8899.384,E2 -8899.384} C_VEL
LIN {X 0,Y 438.995,Z 449.622,A -85,B 0,C 180,E1 -8900.787,E2 -8900.787} C_VEL
LIN {X 0,Y 439.453,Z 442.153,A -85,B 0,C 180,E1 -8902.157,E2 -8902.157} C_VEL
LIN {X 0,Y 439.863,Z 434.188,A -85,B 0,C 180,E1 -8903.348,E2 -8903.348} C_VEL
LIN {X 0,Y 440.511,Z 423.574,A -85,B 0,C 180,E1 -8904.621,E2 -8904.621} C_VEL
LIN {X 0,Y 441.136,Z 412.774,A -85,B 0,C 180,E1 -8905.66,E2 -8905.66} C_VEL
LIN {X 0,Y 441.679,Z 402.284,A -85,B 0,C 180,E1 -8906.465,E2 -8906.465} C_VEL
LIN {X 0,Y 442.282,Z 389.63,A -85,B 0,C 180,E1 -8907.21,E2 -8907.21} C_VEL
LIN {X 0,Y 442.685,Z 376.978,A -85,B 0,C 180,E1 -8907.757,E2 -8907.757} C_VEL
LIN {X 0,Y 443,Z 365.145,A -85,B 0,C 180,E1 -8908.098,E2 -8908.098} C_VEL
LIN {X 0,Y 443.82,Z 277.114,A -85,B 0,C 180,E1 -8909.547,E2 -8909.547} C_VEL
LIN {X 0,Y 440.524,Z 258.581,A -85,B 0,C 180,E1 -8910,E2 -8910} C_VEL
LIN {X 0,Y 440.653,Z 255.006,A -85,B 0,C 180,E1 -8910.685,E2 -8910.685} C_VEL
LIN {X 0,Y 441.3,Z 243.114,A -85,B 0,C 180,E1 -8913.195,E2 -8913.195} C_VEL
LIN {X 0,Y 439.615,Z 232.289,A -85,B 0,C 180,E1 -8915.677,E2 -8915.677} C_VEL
LIN {X 0,Y 439.51,Z 232.24,A -85,B 0,C 180,E1 -8918.274,E2 -8918.274} C_VEL
LIN {X 0,Y 439.447,Z 232.245,A -85,B 0,C 180,E1 -8921.064,E2 -8921.064} C_VEL
LIN {X 0,Y 439.427,Z 232.245,A -85,B 0,C 180,E1 -8923.88,E2 -8923.88} C_VEL
LIN {X 0,Y 439.416,Z 232.252,A -85,B 0,C 180,E1 -8926.731,E2 -8926.731} C_VEL
LIN {X 0,Y 439.395,Z 232.239,A -85,B 0,C 180,E1 -8929.626,E2 -8929.626} C_VEL
LIN {X 0,Y 439.388,Z 232.251,A -85,B 0,C 180,E1 -8932.574,E2 -8932.574} C_VEL
LIN {X 0,Y 439.37,Z 232.238,A -85,B 0,C 180,E1 -8935.587,E2 -8935.587} C_VEL
LIN {X 0,Y 439.397,Z 232.237,A -85,B 0,C 180,E1 -8938.674,E2 -8938.674} C_VEL
LIN {X 0,Y 439.388,Z 232.251,A -85,B 0,C 180,E1 -8942.046,E2 -8942.046} C_VEL
LIN {X 0,Y 439.38,Z 232.249,A -85,B 0,C 180,E1 -8945.348,E2 -8945.348} C_VEL
LIN {X 0,Y 439.402,Z 232.247,A -85,B 0,C 180,E1 -8948.592,E2 -8948.592} C_VEL
LIN {X 0,Y 439.368,Z 232.249,A -85,B 0,C 180,E1 -8951.263,E2 -8951.263} C_VEL
LIN {X 0,Y 439.42,Z 232.243,A -85,B 0,C 180,E1 -8954.726,E2 -8954.726} C_VEL
LIN {X 0,Y 439.384,Z 232.254,A -85,B 0,C 180,E1 -8957.802,E2 -8957.802} C_VEL
LIN {X 0,Y 439.423,Z 232.236,A -85,B 0,C 180,E1 -8960.235,E2 -8960.235} C_VEL
LIN {X 0,Y 439.35,Z 232.248,A -85,B 0,C 180,E1 -8963.718,E2 -8963.718} C_VEL
LIN {X 0,Y 439.349,Z 232.254,A -85,B 0,C 180,E1 -8967.059,E2 -8967.059} C_VEL
LIN {X 0,Y 439.373,Z 232.248,A -85,B 0,C 180,E1 -8970.28,E2 -8970.28} C_VEL
LIN {X 0,Y 439.412,Z 232.232,A -85,B 0,C 180,E1 -8973.593,E2 -8973.593} C_VEL
LIN {X 0,Y 439.37,Z 232.251,A -85,B 0,C 180,E1 -8976.434,E2 -8976.434} C_VEL
LIN {X 0,Y 439.389,Z 232.249,A -85,B 0,C 180,E1 -8979.403,E2 -8979.403} C_VEL
LIN {X 0,Y 439.417,Z 232.238,A -85,B 0,C 180,E1 -8982.314,E2 -8982.314} C_VEL
LIN {X 0,Y 439.435,Z 232.227,A -85,B 0,C 180,E1 -8985.179,E2 -8985.179} C_VEL
LIN {X 0,Y 439.498,Z 232.229,A -85,B 0,C 180,E1 -8988.006,E2 -8988.006} C_VEL
LIN {X 0,Y 439.54,Z 232.232,A -85,B 0,C 180,E1 -8991.731,E2 -8991.731} C_VEL
LIN {X 0,Y 439.617,Z 232.214,A -85,B 0,C 180,E1 -8994.5,E2 -8994.5} C_VEL
LIN {X 0,Y 439.629,Z 232.201,A -85,B 0,C 180,E1 -8998.172,E2 -8998.172} C_VEL
LIN {X 0,Y 439.759,Z 232.199,A -85,B 0,C 180,E1 -9000.004,E2 -9000.004} C_VEL
LIN {X 0,Y 439.638,Z 232.216,A -85,B 0,C 180,E1 -9002.753,E2 -9002.753} C_VEL
LIN {X 0,Y 439.592,Z 232.221,A -85,B 0,C 180,E1 -9006.429,E2 -9006.429} C_VEL
LIN {X 0,Y 439.499,Z 232.221,A -85,B 0,C 180,E1 -9009.205,E2 -9009.205} C_VEL
LIN {X 0,Y 439.468,Z 232.234,A -85,B 0,C 180,E1 -9012.941,E2 -9012.941} C_VEL
LIN {X 0,Y 439.45,Z 232.248,A -85,B 0,C 180,E1 -9016.352,E2 -9016.352} C_VEL
LIN {X 0,Y 439.407,Z 232.238,A -85,B 0,C 180,E1 -9019.629,E2 -9019.629} C_VEL
LIN {X 0,Y 439.369,Z 232.248,A -85,B 0,C 180,E1 -9022.579,E2 -9022.579} C_VEL
LIN {X 0,Y 439.394,Z 232.249,A -85,B 0,C 180,E1 -9025.589,E2 -9025.589} C_VEL
LIN {X 0,Y 439.423,Z 232.244,A -85,B 0,C 180,E1 -9028.676,E2 -9028.676} C_VEL
LIN {X 0,Y 439.372,Z 232.249,A -85,B 0,C 180,E1 -9032.032,E2 -9032.032} C_VEL
LIN {X 0,Y 439.398,Z 232.249,A -85,B 0,C 180,E1 -9035.342,E2 -9035.342} C_VEL
LIN {X 0,Y 439.371,Z 232.249,A -85,B 0,C 180,E1 -9038.599,E2 -9038.599} C_VEL
LIN {X 0,Y 439.39,Z 232.254,A -85,B 0,C 180,E1 -9041.258,E2 -9041.258} C_VEL
LIN {X 0,Y 439.407,Z 232.229,A -85,B 0,C 180,E1 -9044.732,E2 -9044.732} C_VEL
LIN {X 0,Y 439.393,Z 232.251,A -85,B 0,C 180,E1 -9047.796,E2 -9047.796} C_VEL
LIN {X 0,Y 439.368,Z 232.251,A -85,B 0,C 180,E1 -9050.222,E2 -9050.222} C_VEL
LIN {X 0,Y 439.381,Z 232.255,A -85,B 0,C 180,E1 -9053.714,E2 -9053.714} C_VEL
LIN {X 0,Y 439.382,Z 232.251,A -85,B 0,C 180,E1 -9057.055,E2 -9057.055} C_VEL
LIN {X 0,Y 439.389,Z 232.253,A -85,B 0,C 180,E1 -9060.275,E2 -9060.275} C_VEL
LIN {X 0,Y 439.422,Z 232.25,A -85,B 0,C 180,E1 -9063.396,E2 -9063.396} C_VEL
LIN {X 0,Y 439.472,Z 232.464,A -85,B 0,C 180,E1 -9064.483,E2 -9064.483} C_VEL
LIN {X 0,Y 441.649,Z 244.274,A -85,B 0,C 180,E1 -9067.029,E2 -9067.029} C_VEL
LIN {X 0,Y 440.925,Z 259.888,A -85,B 0,C 180,E1 -9070.126,E2 -9070.126} C_VEL
LIN {X 0,Y 440.442,Z 269.582,A -85,B 0,C 180,E1 -9072.001,E2 -9072.001} C_VEL
LIN {X 0,Y 441.25,Z 275.125,A -85,B 0,C 180,E1 -9072.163,E2 -9072.163} C_VEL
LIN {X 0,Y 443.824,Z 291.426,A -85,B 0,C 180,E1 -9072.529,E2 -9072.529} C_VEL
LIN {X 0,Y 442.961,Z 378.103,A -85,B 0,C 180,E1 -9073.969,E2 -9073.969} C_VEL
LIN {X 0,Y 442.545,Z 391.923,A -85,B 0,C 180,E1 -9074.397,E2 -9074.397} C_VEL
LIN {X 0,Y 442.029,Z 404.325,A -85,B 0,C 180,E1 -9074.968,E2 -9074.968} C_VEL
LIN {X 0,Y 441.398,Z 416.205,A -85,B 0,C 180,E1 -9075.713,E2 -9075.713} C_VEL
LIN {X 0,Y 440.862,Z 427.459,A -85,B 0,C 180,E1 -9076.619,E2 -9076.619} C_VEL
LIN {X 0,Y 440.294,Z 437.935,A -85,B 0,C 180,E1 -9077.673,E2 -9077.673} C_VEL
LIN {X 0,Y 439.621,Z 447.985,A -85,B 0,C 180,E1 -9078.94,E2 -9078.94} C_VEL
LIN {X 0,Y 439.116,Z 456.828,A -85,B 0,C 180,E1 -9080.326,E2 -9080.326} C_VEL
LIN {X 0,Y 438.788,Z 463.889,A -85,B 0,C 180,E1 -9081.712,E2 -9081.712} C_VEL
LIN {X 0,Y 438.519,Z 469.524,A -85,B 0,C 180,E1 -9083.097,E2 -9083.097} C_VEL
LIN {X 0,Y 438.408,Z 473.951,A -85,B 0,C 180,E1 -9084.481,E2 -9084.481} C_VEL
LIN {X 0,Y 438.348,Z 476.286,A -85,B 0,C 180,E1 -9085.402,E2 -9085.402} C_VEL
LIN {X 0,Y 438.262,Z 478.191,A -85,B 0,C 180,E1 -9086.323,E2 -9086.323} C_VEL
LIN {X 0,Y 438.297,Z 479.65,A -85,B 0,C 180,E1 -9087.243,E2 -9087.243} C_VEL
LIN {X 0,Y 438.277,Z 480.677,A -85,B 0,C 180,E1 -9088.162,E2 -9088.162} C_VEL
LIN {X 0,Y 438.232,Z 481.569,A -85,B 0,C 180,E1 -9090,E2 -9090} C_VEL
LIN {X 0,Y 438.234,Z 481.409,A -85,B 0,C 180,E1 -9090.919,E2 -9090.919} C_VEL
LIN {X 0,Y 438.277,Z 480.833,A -85,B 0,C 180,E1 -9091.838,E2 -9091.838} C_VEL
LIN {X 0,Y 438.297,Z 479.87,A -85,B 0,C 180,E1 -9092.758,E2 -9092.758} C_VEL
LIN {X 0,Y 438.263,Z 478.514,A -85,B 0,C 180,E1 -9093.678,E2 -9093.678} C_VEL
LIN {X 0,Y 438.424,Z 475.649,A -85,B 0,C 180,E1 -9095.058,E2 -9095.058} C_VEL
LIN {X 0,Y 438.475,Z 471.762,A -85,B 0,C 180,E1 -9096.442,E2 -9096.442} C_VEL
LIN {X 0,Y 438.712,Z 466.755,A -85,B 0,C 180,E1 -9097.826,E2 -9097.826} C_VEL
LIN {X 0,Y 439.095,Z 460.472,A -85,B 0,C 180,E1 -9099.21,E2 -9099.21} C_VEL
LIN {X 0,Y 439.548,Z 452.613,A -85,B 0,C 180,E1 -9100.596,E2 -9100.596} C_VEL
LIN {X 0,Y 440.113,Z 444.614,A -85,B 0,C 180,E1 -9101.748,E2 -9101.748} C_VEL
LIN {X 0,Y 440.736,Z 434.867,A -85,B 0,C 180,E1 -9102.9,E2 -9102.9} C_VEL
LIN {X 0,Y 441.331,Z 424.028,A -85,B 0,C 180,E1 -9103.937,E2 -9103.937} C_VEL
LIN {X 0,Y 442.013,Z 413.427,A -85,B 0,C 180,E1 -9104.738,E2 -9104.738} C_VEL
LIN {X 0,Y 442.697,Z 400.686,A -85,B 0,C 180,E1 -9105.48,E2 -9105.48} C_VEL
LIN {X 0,Y 443.236,Z 387.885,A -85,B 0,C 180,E1 -9106.022,E2 -9106.022} C_VEL
LIN {X 0,Y 443.607,Z 375.379,A -85,B 0,C 180,E1 -9106.362,E2 -9106.362} C_VEL
LIN {X 0,Y 444.396,Z 290.198,A -85,B 0,C 180,E1 -9107.784,E2 -9107.784} C_VEL
LIN {X 0,Y 440.765,Z 269.65,A -85,B 0,C 180,E1 -9108.333,E2 -9108.333} C_VEL
LIN {X 0,Y 440.963,Z 264.394,A -85,B 0,C 180,E1 -9109.312,E2 -9109.312} C_VEL
LIN {X 0,Y 442.022,Z 247.183,A -85,B 0,C 180,E1 -9112.749,E2 -9112.749} C_VEL
LIN {X 0,Y 441.556,Z 242.723,A -85,B 0,C 180,E1 -9113.697,E2 -9113.697} C_VEL
LIN {X 0,Y 439.439,Z 232.338,A -85,B 0,C 180,E1 -9116.066,E2 -9116.066} C_VEL
LIN {X 0,Y 439.429,Z 232.247,A -85,B 0,C 180,E1 -9118.673,E2 -9118.673} C_VEL
LIN {X 0,Y 439.381,Z 232.256,A -85,B 0,C 180,E1 -9122.029,E2 -9122.029} C_VEL
LIN {X 0,Y 439.404,Z 232.248,A -85,B 0,C 180,E1 -9125.339,E2 -9125.339} C_VEL
LIN {X 0,Y 439.373,Z 232.249,A -85,B 0,C 180,E1 -9128.596,E2 -9128.596} C_VEL
LIN {X 0,Y 439.394,Z 232.247,A -85,B 0,C 180,E1 -9132.205,E2 -9132.205} C_VEL
LIN {X 0,Y 439.388,Z 232.25,A -85,B 0,C 180,E1 -9135.266,E2 -9135.266} C_VEL
LIN {X 0,Y 439.393,Z 232.25,A -85,B 0,C 180,E1 -9138.743,E2 -9138.743} C_VEL
LIN {X 0,Y 439.376,Z 232.248,A -85,B 0,C 180,E1 -9141.608,E2 -9141.608} C_VEL
LIN {X 0,Y 439.406,Z 232.25,A -85,B 0,C 180,E1 -9144.841,E2 -9144.841} C_VEL
LIN {X 0,Y 439.38,Z 232.247,A -85,B 0,C 180,E1 -9148.137,E2 -9148.137} C_VEL
LIN {X 0,Y 439.41,Z 232.244,A -85,B 0,C 180,E1 -9151.604,E2 -9151.604} C_VEL
LIN {X 0,Y 439.375,Z 232.251,A -85,B 0,C 180,E1 -9154.41,E2 -9154.41} C_VEL
LIN {X 0,Y 439.371,Z 232.257,A -85,B 0,C 180,E1 -9157.422,E2 -9157.422} C_VEL
LIN {X 0,Y 439.449,Z 232.237,A -85,B 0,C 180,E1 -9160.66,E2 -9160.66} C_VEL
LIN {X 0,Y 439.47,Z 232.233,A -85,B 0,C 180,E1 -9164.221,E2 -9164.221} C_VEL
LIN {X 0,Y 439.489,Z 232.235,A -85,B 0,C 180,E1 -9167.998,E2 -9167.998} C_VEL
LIN {X 0,Y 439.507,Z 232.242,A -85,B 0,C 180,E1 -9171.722,E2 -9171.722} C_VEL
LIN {X 0,Y 439.613,Z 232.22,A -85,B 0,C 180,E1 -9174.492,E2 -9174.492} C_VEL
LIN {X 0,Y 439.631,Z 232.218,A -85,B 0,C 180,E1 -9178.164,E2 -9178.164} C_VEL
LIN {X 0,Y 439.759,Z 232.206,A -85,B 0,C 180,E1 -9179.996,E2 -9179.996} C_VEL
LIN {X 0,Y 439.63,Z 232.214,A -85,B 0,C 180,E1 -9182.745,E2 -9182.745} C_VEL
LIN {X 0,Y 439.588,Z 232.225,A -85,B 0,C 180,E1 -9186.421,E2 -9186.421} C_VEL
LIN {X 0,Y 439.491,Z 232.237,A -85,B 0,C 180,E1 -9189.197,E2 -9189.197} C_VEL
LIN {X 0,Y 439.459,Z 232.243,A -85,B 0,C 180,E1 -9192.933,E2 -9192.933} C_VEL
LIN {X 0,Y 439.437,Z 232.244,A -85,B 0,C 180,E1 -9196.343,E2 -9196.343} C_VEL
LIN {X 0,Y 439.39,Z 232.249,A -85,B 0,C 180,E1 -9199.621,E2 -9199.621} C_VEL
LIN {X 0,Y 439.352,Z 232.255,A -85,B 0,C 180,E1 -9202.571,E2 -9202.571} C_VEL
LIN {X 0,Y 439.388,Z 232.24,A -85,B 0,C 180,E1 -9205.58,E2 -9205.58} C_VEL
LIN {X 0,Y 439.398,Z 232.251,A -85,B 0,C 180,E1 -9208.669,E2 -9208.669} C_VEL
LIN {X 0,Y 439.348,Z 232.253,A -85,B 0,C 180,E1 -9212.026,E2 -9212.026} C_VEL
LIN {X 0,Y 439.372,Z 232.251,A -85,B 0,C 180,E1 -9215.336,E2 -9215.336} C_VEL
LIN {X 0,Y 439.374,Z 232.248,A -85,B 0,C 180,E1 -9218.589,E2 -9218.589} C_VEL
LIN {X 0,Y 439.377,Z 232.252,A -85,B 0,C 180,E1 -9221.255,E2 -9221.255} C_VEL
LIN {X 0,Y 439.378,Z 232.253,A -85,B 0,C 180,E1 -9224.724,E2 -9224.724} C_VEL
LIN {X 0,Y 439.428,Z 232.374,A -85,B 0,C 180,E1 -9228.161,E2 -9228.161} C_VEL
LIN {X 0,Y 441.378,Z 242.265,A -85,B 0,C 180,E1 -9230.438,E2 -9230.438} C_VEL
LIN {X 0,Y 441.329,Z 247.834,A -85,B 0,C 180,E1 -9231.606,E2 -9231.606} C_VEL
LIN {X 0,Y 440.877,Z 258.233,A -85,B 0,C 180,E1 -9233.705,E2 -9233.705} C_VEL
LIN {X 0,Y 444.563,Z 277.174,A -85,B 0,C 180,E1 -9234.24,E2 -9234.24} C_VEL
LIN {X 0,Y 443.575,Z 366.372,A -85,B 0,C 180,E1 -9235.739,E2 -9235.739} C_VEL
LIN {X 0,Y 443.203,Z 379.813,A -85,B 0,C 180,E1 -9236.16,E2 -9236.16} C_VEL
LIN {X 0,Y 442.706,Z 392.034,A -85,B 0,C 180,E1 -9236.723,E2 -9236.723} C_VEL
LIN {X 0,Y 442.049,Z 404.37,A -85,B 0,C 180,E1 -9237.499,E2 -9237.499} C_VEL
LIN {X 0,Y 441.429,Z 415.881,A -85,B 0,C 180,E1 -9238.439,E2 -9238.439} C_VEL
LIN {X 0,Y 440.753,Z 425.591,A -85,B 0,C 180,E1 -9239.423,E2 -9239.423} C_VEL
LIN {X 0,Y 440.123,Z 434.941,A -85,B 0,C 180,E1 -9240.592,E2 -9240.592} C_VEL
LIN {X 0,Y 439.548,Z 443.253,A -85,B 0,C 180,E1 -9241.87,E2 -9241.87} C_VEL
LIN {X 0,Y 439.035,Z 451.112,A -85,B 0,C 180,E1 -9243.37,E2 -9243.37} C_VEL
LIN {X 0,Y 438.705,Z 457.293,A -85,B 0,C 180,E1 -9244.879,E2 -9244.879} C_VEL
LIN {X 0,Y 438.467,Z 462.022,A -85,B 0,C 180,E1 -9246.377,E2 -9246.377} C_VEL
LIN {X 0,Y 438.357,Z 464.478,A -85,B 0,C 180,E1 -9247.37,E2 -9247.37} C_VEL
LIN {X 0,Y 438.26,Z 466.532,A -85,B 0,C 180,E1 -9248.432,E2 -9248.432} C_VEL
LIN {X 0,Y 438.153,Z 468.485,A -85,B 0,C 180,E1 -9249.99,E2 -9249.99} C_VEL
LIN {X 0,Y 437.448,Z 469.123,A -85,B 0,C 180,E1 -9250.753,E2 -9250.753} C_VEL
LIN {X 0,Y 434.515,Z 469.488,A -85,B 0,C 180,E1 -9251.997,E2 -9251.997} C_VEL
LIN {X 0,Y 432.099,Z 469.23,A -85,B 0,C 180,E1 -9253.003,E2 -9253.003} C_VEL
LIN {X 0,Y 431.137,Z 468.728,A -85,B 0,C 180,E1 -9253.778,E2 -9253.778} C_VEL
LIN {X 0,Y 431.099,Z 468.495,A -85,B 0,C 180,E1 -9254.04,E2 -9254.04} C_VEL
LIN {X 0,Y 431.13,Z 467.525,A -85,B 0,C 180,E1 -9254.881,E2 -9254.881} C_VEL
LIN {X 0,Y 431.229,Z 465.042,A -85,B 0,C 180,E1 -9256.331,E2 -9256.331} C_VEL
LIN {X 0,Y 431.414,Z 461.522,A -85,B 0,C 180,E1 -9257.773,E2 -9257.773} C_VEL
LIN {X 0,Y 431.607,Z 456.887,A -85,B 0,C 180,E1 -9259.207,E2 -9259.207} C_VEL
LIN {X 0,Y 431.954,Z 449.854,A -85,B 0,C 180,E1 -9260.872,E2 -9260.872} C_VEL
LIN {X 0,Y 432.463,Z 441.661,A -85,B 0,C 180,E1 -9262.392,E2 -9262.392} C_VEL
LIN {X 0,Y 432.997,Z 432.706,A -85,B 0,C 180,E1 -9263.71,E2 -9263.71} C_VEL
LIN {X 0,Y 433.6,Z 422.85,A -85,B 0,C 180,E1 -9264.885,E2 -9264.885} C_VEL
LIN {X 0,Y 434.159,Z 413.187,A -85,B 0,C 180,E1 -9265.822,E2 -9265.822} C_VEL
LIN {X 0,Y 434.736,Z 402.78,A -85,B 0,C 180,E1 -9266.64,E2 -9266.64} C_VEL
LIN {X 0,Y 435.303,Z 391.184,A -85,B 0,C 180,E1 -9267.351,E2 -9267.351} C_VEL
LIN {X 0,Y 435.778,Z 378.028,A -85,B 0,C 180,E1 -9267.943,E2 -9267.943} C_VEL
LIN {X 0,Y 436.137,Z 365.058,A -85,B 0,C 180,E1 -9268.33,E2 -9268.33} C_VEL
LIN {X 0,Y 437.018,Z 277.918,A -85,B 0,C 180,E1 -9269.788,E2 -9269.788} C_VEL
LIN {X 0,Y 433.589,Z 258.663,A -85,B 0,C 180,E1 -9270.261,E2 -9270.261} C_VEL
LIN {X 0,Y 433.833,Z 253.059,A -85,B 0,C 180,E1 -9271.392,E2 -9271.392} C_VEL
LIN {X 0,Y 434.241,Z 243.356,A -85,B 0,C 180,E1 -9273.479,E2 -9273.479} C_VEL
LIN {X 0,Y 432.573,Z 233.172,A -85,B 0,C 180,E1 -9275.857,E2 -9275.857} C_VEL
LIN {X 0,Y 432.47,Z 233.114,A -85,B 0,C 180,E1 -9279.352,E2 -9279.352} C_VEL
LIN {X 0,Y 432.449,Z 233.116,A -85,B 0,C 180,E1 -9283.151,E2 -9283.151} C_VEL
LIN {X 0,Y 432.396,Z 233.125,A -85,B 0,C 180,E1 -9286.495,E2 -9286.495} C_VEL
LIN {X 0,Y 432.344,Z 233.117,A -85,B 0,C 180,E1 -9289.96,E2 -9289.96} C_VEL
LIN {X 0,Y 432.32,Z 233.137,A -85,B 0,C 180,E1 -9292.964,E2 -9292.964} C_VEL
LIN {X 0,Y 432.321,Z 233.113,A -85,B 0,C 180,E1 -9296.035,E2 -9296.035} C_VEL
LIN {X 0,Y 432.324,Z 233.123,A -85,B 0,C 180,E1 -9299.188,E2 -9299.188} C_VEL
LIN {X 0,Y 432.327,Z 233.13,A -85,B 0,C 180,E1 -9302.306,E2 -9302.306} C_VEL
LIN {X 0,Y 432.329,Z 233.124,A -85,B 0,C 180,E1 -9304.677,E2 -9304.677} C_VEL
LIN {X 0,Y 432.348,Z 233.128,A -85,B 0,C 180,E1 -9308.148,E2 -9308.148} C_VEL
LIN {X 0,Y 432.339,Z 233.122,A -85,B 0,C 180,E1 -9311.796,E2 -9311.796} C_VEL
LIN {X 0,Y 432.371,Z 233.123,A -85,B 0,C 180,E1 -9314.349,E2 -9314.349} C_VEL
LIN {X 0,Y 432.343,Z 233.126,A -85,B 0,C 180,E1 -9317.012,E2 -9317.012} C_VEL
LIN {X 0,Y 432.329,Z 233.127,A -85,B 0,C 180,E1 -9319.821,E2 -9319.821} C_VEL
LIN {X 0,Y 432.29,Z 233.125,A -85,B 0,C 180,E1 -9323.028,E2 -9323.028} C_VEL
LIN {X 0,Y 432.333,Z 233.13,A -85,B 0,C 180,E1 -9326.001,E2 -9326.001} C_VEL
LIN {X 0,Y 432.371,Z 233.117,A -85,B 0,C 180,E1 -9329.749,E2 -9329.749} C_VEL
LIN {X 0,Y 432.379,Z 233.108,A -85,B 0,C 180,E1 -9333.377,E2 -9333.377} C_VEL
LIN {X 0,Y 432.354,Z 233.121,A -85,B 0,C 180,E1 -9336.028,E2 -9336.028} C_VEL
LIN {X 0,Y 432.351,Z 233.129,A -85,B 0,C 180,E1 -9339.052,E2 -9339.052} C_VEL
LIN {X 0,Y 432.364,Z 233.115,A -85,B 0,C 180,E1 -9342.016,E2 -9342.016} C_VEL
LIN {X 0,Y 432.382,Z 233.103,A -85,B 0,C 180,E1 -9344.931,E2 -9344.931} C_VEL
LIN {X 0,Y 432.471,Z 233.105,A -85,B 0,C 180,E1 -9347.809,E2 -9347.809} C_VEL
LIN {X 0,Y 432.484,Z 233.112,A -85,B 0,C 180,E1 -9351.595,E2 -9351.595} C_VEL
LIN {X 0,Y 432.593,Z 233.088,A -85,B 0,C 180,E1 -9354.411,E2 -9354.411} C_VEL
LIN {X 0,Y 432.599,Z 233.077,A -85,B 0,C 180,E1 -9358.142,E2 -9358.142} C_VEL
LIN {X 0,Y 432.728,Z 233.074,A -85,B 0,C 180,E1 -9360.004,E2 -9360.004} C_VEL
LIN {X 0,Y 432.59,Z 233.094,A -85,B 0,C 180,E1 -9362.798,E2 -9362.798} C_VEL
LIN {X 0,Y 432.586,Z 233.1,A -85,B 0,C 180,E1 -9365.598,E2 -9365.598} C_VEL
LIN {X 0,Y 432.483,Z 233.097,A -85,B 0,C 180,E1 -9368.414,E2 -9368.414} C_VEL
LIN {X 0,Y 432.461,Z 233.105,A -85,B 0,C 180,E1 -9372.2,E2 -9372.2} C_VEL
LIN {X 0,Y 432.434,Z 233.119,A -85,B 0,C 180,E1 -9376.042,E2 -9376.042} C_VEL
LIN {X 0,Y 432.391,Z 233.112,A -85,B 0,C 180,E1 -9379.488,E2 -9379.488} C_VEL
LIN {X 0,Y 432.323,Z 233.129,A -85,B 0,C 180,E1 -9382.967,E2 -9382.967} C_VEL
LIN {X 0,Y 432.348,Z 233.13,A -85,B 0,C 180,E1 -9385.005,E2 -9385.005} C_VEL
LIN {X 0,Y 432.387,Z 233.119,A -85,B 0,C 180,E1 -9388.126,E2 -9388.126} C_VEL
LIN {X 0,Y 432.326,Z 233.13,A -85,B 0,C 180,E1 -9391.349,E2 -9391.349} C_VEL
LIN {X 0,Y 432.335,Z 233.132,A -85,B 0,C 180,E1 -9394.681,E2 -9394.681} C_VEL
LIN {X 0,Y 432.338,Z 233.123,A -85,B 0,C 180,E1 -9398.153,E2 -9398.153} C_VEL
LIN {X 0,Y 432.333,Z 233.128,A -85,B 0,C 180,E1 -9401.603,E2 -9401.603} C_VEL
LIN {X 0,Y 432.343,Z 233.108,A -85,B 0,C 180,E1 -9404.349,E2 -9404.349} C_VEL
LIN {X 0,Y 432.325,Z 233.119,A -85,B 0,C 180,E1 -9407.018,E2 -9407.018} C_VEL
LIN {X 0,Y 432.323,Z 233.133,A -85,B 0,C 180,E1 -9409.826,E2 -9409.826} C_VEL
LIN {X 0,Y 432.313,Z 233.128,A -85,B 0,C 180,E1 -9413.023,E2 -9413.023} C_VEL
LIN {X 0,Y 432.369,Z 233.126,A -85,B 0,C 180,E1 -9415.998,E2 -9415.998} C_VEL
LIN {X 0,Y 432.356,Z 233.128,A -85,B 0,C 180,E1 -9419.491,E2 -9419.491} C_VEL
LIN {X 0,Y 432.381,Z 233.129,A -85,B 0,C 180,E1 -9421.877,E2 -9421.877} C_VEL
LIN {X 0,Y 432.437,Z 233.203,A -85,B 0,C 180,E1 -9424.232,E2 -9424.232} C_VEL
LIN {X 0,Y 433.652,Z 239.69,A -85,B 0,C 180,E1 -9425.7,E2 -9425.7} C_VEL
LIN {X 0,Y 434.705,Z 246.561,A -85,B 0,C 180,E1 -9427.169,E2 -9427.169} C_VEL
LIN {X 0,Y 433.789,Z 263.648,A -85,B 0,C 180,E1 -9430.602,E2 -9430.602} C_VEL
LIN {X 0,Y 433.469,Z 269.689,A -85,B 0,C 180,E1 -9431.756,E2 -9431.756} C_VEL
LIN {X 0,Y 436.985,Z 292.333,A -85,B 0,C 180,E1 -9432.298,E2 -9432.298} C_VEL
LIN {X 0,Y 436.101,Z 377.954,A -85,B 0,C 180,E1 -9433.74,E2 -9433.74} C_VEL
LIN {X 0,Y 435.649,Z 391.787,A -85,B 0,C 180,E1 -9434.173,E2 -9434.173} C_VEL
LIN {X 0,Y 435.082,Z 404.706,A -85,B 0,C 180,E1 -9434.782,E2 -9434.782} C_VEL
LIN {X 0,Y 434.429,Z 417.281,A -85,B 0,C 180,E1 -9435.598,E2 -9435.598} C_VEL
LIN {X 0,Y 433.821,Z 428.987,A -85,B 0,C 180,E1 -9436.581,E2 -9436.581} C_VEL
LIN {X 0,Y 433.24,Z 438.567,A -85,B 0,C 180,E1 -9437.588,E2 -9437.588} C_VEL
LIN {X 0,Y 432.634,Z 447.674,A -85,B 0,C 180,E1 -9438.759,E2 -9438.759} C_VEL
LIN {X 0,Y 432.094,Z 456.553,A -85,B 0,C 180,E1 -9440.167,E2 -9440.167} C_VEL
LIN {X 0,Y 431.722,Z 463.659,A -85,B 0,C 180,E1 -9441.576,E2 -9441.576} C_VEL
LIN {X 0,Y 431.44,Z 469.322,A -85,B 0,C 180,E1 -9442.983,E2 -9442.983} C_VEL
LIN {X 0,Y 431.31,Z 473.775,A -85,B 0,C 180,E1 -9444.39,E2 -9444.39} C_VEL
LIN {X 0,Y 431.279,Z 476.124,A -85,B 0,C 180,E1 -9445.327,E2 -9445.327} C_VEL
LIN {X 0,Y 431.172,Z 478.039,A -85,B 0,C 180,E1 -9446.262,E2 -9446.262} C_VEL
LIN {X 0,Y 431.193,Z 479.518,A -85,B 0,C 180,E1 -9447.198,E2 -9447.198} C_VEL
LIN {X 0,Y 431.201,Z 480.556,A -85,B 0,C 180,E1 -9448.132,E2 -9448.132} C_VEL
LIN {X 0,Y 431.148,Z 481.466,A -85,B 0,C 180,E1 -9450,E2 -9450} C_VEL
LIN {X 0,Y 431.152,Z 481.325,A -85,B 0,C 180,E1 -9450.934,E2 -9450.934} C_VEL
LIN {X 0,Y 431.201,Z 480.759,A -85,B 0,C 180,E1 -9451.868,E2 -9451.868} C_VEL
LIN {X 0,Y 431.193,Z 479.805,A -85,B 0,C 180,E1 -9452.803,E2 -9452.803} C_VEL
LIN {X 0,Y 431.172,Z 478.459,A -85,B 0,C 180,E1 -9453.739,E2 -9453.739} C_VEL
LIN {X 0,Y 431.336,Z 475.615,A -85,B 0,C 180,E1 -9455.142,E2 -9455.142} C_VEL
LIN {X 0,Y 431.394,Z 471.75,A -85,B 0,C 180,E1 -9456.549,E2 -9456.549} C_VEL
LIN {X 0,Y 431.662,Z 466.765,A -85,B 0,C 180,E1 -9457.955,E2 -9457.955} C_VEL
LIN {X 0,Y 432.043,Z 460.511,A -85,B 0,C 180,E1 -9459.362,E2 -9459.362} C_VEL
LIN {X 0,Y 432.551,Z 452.693,A -85,B 0,C 180,E1 -9460.769,E2 -9460.769} C_VEL
LIN {X 0,Y 433.172,Z 444.728,A -85,B 0,C 180,E1 -9461.939,E2 -9461.939} C_VEL
LIN {X 0,Y 433.823,Z 435.024,A -85,B 0,C 180,E1 -9463.109,E2 -9463.109} C_VEL
LIN {X 0,Y 434.452,Z 424.255,A -85,B 0,C 180,E1 -9464.163,E2 -9464.163} C_VEL
LIN {X 0,Y 435.157,Z 413.774,A -85,B 0,C 180,E1 -9464.976,E2 -9464.976} C_VEL
LIN {X 0,Y 435.896,Z 401.178,A -85,B 0,C 180,E1 -9465.728,E2 -9465.728} C_VEL
LIN {X 0,Y 436.494,Z 387.855,A -85,B 0,C 180,E1 -9466.306,E2 -9466.306} C_VEL
LIN {X 0,Y 436.893,Z 375.438,A -85,B 0,C 180,E1 -9466.651,E2 -9466.651} C_VEL
LIN {X 0,Y 437.687,Z 290.818,A -85,B 0,C 180,E1 -9468.09,E2 -9468.09} C_VEL
LIN {X 0,Y 433.902,Z 269.709,A -85,B 0,C 180,E1 -9468.667,E2 -9468.667} C_VEL
LIN {X 0,Y 433.906,Z 268.106,A -85,B 0,C 180,E1 -9468.902,E2 -9468.902} C_VEL
LIN {X 0,Y 435.005,Z 250.045,A -85,B 0,C 180,E1 -9472.564,E2 -9472.564} C_VEL
LIN {X 0,Y 435.01,Z 246.424,A -85,B 0,C 180,E1 -9473.321,E2 -9473.321} C_VEL
LIN {X 0,Y 432.676,Z 234.488,A -85,B 0,C 180,E1 -9476.012,E2 -9476.012} C_VEL
LIN {X 0,Y 432.406,Z 233.144,A -85,B 0,C 180,E1 -9476.429,E2 -9476.429} C_VEL
LIN {X 0,Y 432.354,Z 233.127,A -85,B 0,C 180,E1 -9479.187,E2 -9479.187} C_VEL
LIN {X 0,Y 432.335,Z 233.128,A -85,B 0,C 180,E1 -9482.442,E2 -9482.442} C_VEL
LIN {X 0,Y 432.355,Z 233.125,A -85,B 0,C 180,E1 -9485.63,E2 -9485.63} C_VEL
LIN {X 0,Y 432.336,Z 233.125,A -85,B 0,C 180,E1 -9488.71,E2 -9488.71} C_VEL
LIN {X 0,Y 432.332,Z 233.13,A -85,B 0,C 180,E1 -9491.797,E2 -9491.797} C_VEL
LIN {X 0,Y 432.344,Z 233.13,A -85,B 0,C 180,E1 -9494.346,E2 -9494.346} C_VEL
LIN {X 0,Y 432.328,Z 233.119,A -85,B 0,C 180,E1 -9497.015,E2 -9497.015} C_VEL
LIN {X 0,Y 432.325,Z 233.13,A -85,B 0,C 180,E1 -9499.822,E2 -9499.822} C_VEL
LIN {X 0,Y 432.315,Z 233.135,A -85,B 0,C 180,E1 -9503.02,E2 -9503.02} C_VEL
LIN {X 0,Y 432.344,Z 233.127,A -85,B 0,C 180,E1 -9506,E2 -9506} C_VEL
LIN {X 0,Y 432.357,Z 233.127,A -85,B 0,C 180,E1 -9509.488,E2 -9509.488} C_VEL
LIN {X 0,Y 432.337,Z 233.123,A -85,B 0,C 180,E1 -9511.87,E2 -9511.87} C_VEL
LIN {X 0,Y 432.363,Z 233.123,A -85,B 0,C 180,E1 -9515.543,E2 -9515.543} C_VEL
LIN {X 0,Y 432.359,Z 233.13,A -85,B 0,C 180,E1 -9519.043,E2 -9519.043} C_VEL
LIN {X 0,Y 432.369,Z 233.125,A -85,B 0,C 180,E1 -9522.007,E2 -9522.007} C_VEL
LIN {X 0,Y 432.401,Z 233.114,A -85,B 0,C 180,E1 -9524.923,E2 -9524.923} C_VEL
LIN {X 0,Y 432.465,Z 233.113,A -85,B 0,C 180,E1 -9527.8,E2 -9527.8} C_VEL
LIN {X 0,Y 432.467,Z 233.117,A -85,B 0,C 180,E1 -9531.586,E2 -9531.586} C_VEL
LIN {X 0,Y 432.589,Z 233.095,A -85,B 0,C 180,E1 -9534.402,E2 -9534.402} C_VEL
LIN {X 0,Y 432.601,Z 233.093,A -85,B 0,C 180,E1 -9538.134,E2 -9538.134} C_VEL
LIN {X 0,Y 432.728,Z 233.082,A -85,B 0,C 180,E1 -9539.996,E2 -9539.996} C_VEL
LIN {X 0,Y 432.582,Z 233.092,A -85,B 0,C 180,E1 -9542.789,E2 -9542.789} C_VEL
LIN {X 0,Y 432.582,Z 233.098,A -85,B 0,C 180,E1 -9545.59,E2 -9545.59} C_VEL
LIN {X 0,Y 432.459,Z 233.115,A -85,B 0,C 180,E1 -9548.406,E2 -9548.406} C_VEL
LIN {X 0,Y 432.452,Z 233.112,A -85,B 0,C 180,E1 -9552.192,E2 -9552.192} C_VEL
LIN {X 0,Y 432.421,Z 233.115,A -85,B 0,C 180,E1 -9556.034,E2 -9556.034} C_VEL
LIN {X 0,Y 432.375,Z 233.123,A -85,B 0,C 180,E1 -9559.48,E2 -9559.48} C_VEL
LIN {X 0,Y 432.306,Z 233.137,A -85,B 0,C 180,E1 -9562.959,E2 -9562.959} C_VEL
LIN {X 0,Y 432.347,Z 233.115,A -85,B 0,C 180,E1 -9566.028,E2 -9566.028} C_VEL
LIN {X 0,Y 432.323,Z 233.134,A -85,B 0,C 180,E1 -9569.183,E2 -9569.183} C_VEL
LIN {X 0,Y 432.301,Z 233.132,A -85,B 0,C 180,E1 -9572.438,E2 -9572.438} C_VEL
LIN {X 0,Y 432.321,Z 233.131,A -85,B 0,C 180,E1 -9575.627,E2 -9575.627} C_VEL
LIN {X 0,Y 432.342,Z 233.131,A -85,B 0,C 180,E1 -9579.336,E2 -9579.336} C_VEL
LIN {X 0,Y 432.345,Z 233.133,A -85,B 0,C 180,E1 -9581.788,E2 -9581.788} C_VEL
LIN {X 0,Y 432.348,Z 233.13,A -85,B 0,C 180,E1 -9584.337,E2 -9584.337} C_VEL
LIN {X 0,Y 432.366,Z 233.239,A -85,B 0,C 180,E1 -9587.863,E2 -9587.863} C_VEL
LIN {X 0,Y 434.141,Z 241.769,A -85,B 0,C 180,E1 -9589.887,E2 -9589.887} C_VEL
LIN {X 0,Y 434.565,Z 246.41,A -85,B 0,C 180,E1 -9590.911,E2 -9590.911} C_VEL
LIN {X 0,Y 434.022,Z 258.286,A -85,B 0,C 180,E1 -9593.354,E2 -9593.354} C_VEL
LIN {X 0,Y 434.931,Z 262.851,A -85,B 0,C 180,E1 -9593.523,E2 -9593.523} C_VEL
LIN {X 0,Y 437.874,Z 277.91,A -85,B 0,C 180,E1 -9593.933,E2 -9593.933} C_VEL
LIN {X 0,Y 436.891,Z 365.902,A -85,B 0,C 180,E1 -9595.433,E2 -9595.433} C_VEL
LIN {X 0,Y 436.487,Z 378.983,A -85,B 0,C 180,E1 -9595.838,E2 -9595.838} C_VEL
LIN {X 0,Y 435.954,Z 391.562,A -85,B 0,C 180,E1 -9596.416,E2 -9596.416} C_VEL
LIN {X 0,Y 435.28,Z 403.707,A -85,B 0,C 180,E1 -9597.178,E2 -9597.178} C_VEL
LIN {X 0,Y 434.585,Z 415.613,A -85,B 0,C 180,E1 -9598.156,E2 -9598.156} C_VEL
LIN {X 0,Y 433.82,Z 426.103,A -85,B 0,C 180,E1 -9599.236,E2 -9599.236} C_VEL
LIN {X 0,Y 433.195,Z 434.798,A -85,B 0,C 180,E1 -9600.342,E2 -9600.342} C_VEL
LIN {X 0,Y 432.634,Z 442.766,A -85,B 0,C 180,E1 -9601.574,E2 -9601.574} C_VEL
LIN {X 0,Y 432.106,Z 449.836,A -85,B 0,C 180,E1 -9602.909,E2 -9602.909} C_VEL
LIN {X 0,Y 431.713,Z 456.335,A -85,B 0,C 180,E1 -9604.443,E2 -9604.443} C_VEL
LIN {X 0,Y 431.449,Z 461.352,A -85,B 0,C 180,E1 -9605.969,E2 -9605.969} C_VEL
LIN {X 0,Y 431.264,Z 465.056,A -85,B 0,C 180,E1 -9607.482,E2 -9607.482} C_VEL
LIN {X 0,Y 431.139,Z 467.595,A -85,B 0,C 180,E1 -9608.984,E2 -9608.984} C_VEL
LIN {X 0,Y 431.084,Z 468.673,A -85,B 0,C 180,E1 -9609.979,E2 -9609.979} C_VEL
LIN {X 0,Y 431.06,Z 469.339,A -85,B 0,C 180,E1 -9610.999,E2 -9610.999} C_VEL
LIN {X 0,Y 431.041,Z 469.54,A -85,B 0,C 180,E1 -9611.953,E2 -9611.953} C_VEL
LIN {X 0,Y 431.038,Z 469.28,A -85,B 0,C 180,E1 -9612.933,E2 -9612.933} C_VEL
LIN {X 0,Y 431.099,Z 468.495,A -85,B 0,C 180,E1 -9614.04,E2 -9614.04} C_VEL
LIN {X 0,Y 430.54,Z 467.673,A -85,B 0,C 180,E1 -9614.813,E2 -9614.813} C_VEL
LIN {X 0,Y 427.747,Z 465.717,A -85,B 0,C 180,E1 -9616.056,E2 -9616.056} C_VEL
LIN {X 0,Y 425.365,Z 463.621,A -85,B 0,C 180,E1 -9617.043,E2 -9617.043} C_VEL
LIN {X 0,Y 424.397,Z 461.738,A -85,B 0,C 180,E1 -9617.792,E2 -9617.792} C_VEL
LIN {X 0,Y 424.351,Z 461.011,A -85,B 0,C 180,E1 -9618.043,E2 -9618.043} C_VEL
LIN {X 0,Y 424.554,Z 456.185,A -85,B 0,C 180,E1 -9619.508,E2 -9619.508} C_VEL
LIN {X 0,Y 424.893,Z 450.09,A -85,B 0,C 180,E1 -9620.959,E2 -9620.959} C_VEL
LIN {X 0,Y 425.401,Z 442.502,A -85,B 0,C 180,E1 -9622.405,E2 -9622.405} C_VEL
LIN {X 0,Y 425.822,Z 434.788,A -85,B 0,C 180,E1 -9623.603,E2 -9623.603} C_VEL
LIN {X 0,Y 426.441,Z 425.368,A -85,B 0,C 180,E1 -9624.799,E2 -9624.799} C_VEL
LIN {X 0,Y 427.115,Z 414.879,A -85,B 0,C 180,E1 -9625.871,E2 -9625.871} C_VEL
LIN {X 0,Y 427.796,Z 403.231,A -85,B 0,C 180,E1 -9626.821,E2 -9626.821} C_VEL
LIN {X 0,Y 428.443,Z 390.846,A -85,B 0,C 180,E1 -9627.591,E2 -9627.591} C_VEL
LIN {X 0,Y 428.922,Z 377.926,A -85,B 0,C 180,E1 -9628.177,E2 -9628.177} C_VEL
LIN {X 0,Y 429.28,Z 365.297,A -85,B 0,C 180,E1 -9628.559,E2 -9628.559} C_VEL
LIN {X 0,Y 430.174,Z 278.656,A -85,B 0,C 180,E1 -9630.034,E2 -9630.034} C_VEL
LIN {X 0,Y 426.628,Z 258.764,A -85,B 0,C 180,E1 -9630.531,E2 -9630.531} C_VEL
LIN {X 0,Y 426.868,Z 253.269,A -85,B 0,C 180,E1 -9631.651,E2 -9631.651} C_VEL
LIN {X 0,Y 427.281,Z 244.642,A -85,B 0,C 180,E1 -9633.536,E2 -9633.536} C_VEL
LIN {X 0,Y 425.528,Z 234.057,A -85,B 0,C 180,E1 -9636.043,E2 -9636.043} C_VEL
LIN {X 0,Y 425.43,Z 233.993,A -85,B 0,C 180,E1 -9638.55,E2 -9638.55} C_VEL
LIN {X 0,Y 425.433,Z 233.991,A -85,B 0,C 180,E1 -9642.401,E2 -9642.401} C_VEL
LIN {X 0,Y 425.365,Z 233.999,A -85,B 0,C 180,E1 -9646.312,E2 -9646.312} C_VEL
LIN {X 0,Y 425.33,Z 233.991,A -85,B 0,C 180,E1 -9649.656,E2 -9649.656} C_VEL
LIN {X 0,Y 425.32,Z 234.002,A -85,B 0,C 180,E1 -9652.336,E2 -9652.336} C_VEL
LIN {X 0,Y 425.256,Z 233.996,A -85,B 0,C 180,E1 -9655.447,E2 -9655.447} C_VEL
LIN {X 0,Y 425.31,Z 233.99,A -85,B 0,C 180,E1 -9658.633,E2 -9658.633} C_VEL
LIN {X 0,Y 425.3,Z 234.007,A -85,B 0,C 180,E1 -9661.923,E2 -9661.923} C_VEL
LIN {X 0,Y 425.28,Z 234.004,A -85,B 0,C 180,E1 -9665.337,E2 -9665.337} C_VEL
LIN {X 0,Y 425.313,Z 234.003,A -85,B 0,C 180,E1 -9668.896,E2 -9668.896} C_VEL
LIN {X 0,Y 425.303,Z 233.992,A -85,B 0,C 180,E1 -9672.649,E2 -9672.649} C_VEL
LIN {X 0,Y 425.322,Z 234.007,A -85,B 0,C 180,E1 -9676.06,E2 -9676.06} C_VEL
LIN {X 0,Y 425.279,Z 234.003,A -85,B 0,C 180,E1 -9678.63,E2 -9678.63} C_VEL
LIN {X 0,Y 425.296,Z 233.988,A -85,B 0,C 180,E1 -9681.109,E2 -9681.109} C_VEL
LIN {X 0,Y 425.274,Z 234.009,A -85,B 0,C 180,E1 -9684.669,E2 -9684.669} C_VEL
LIN {X 0,Y 425.249,Z 234.013,A -85,B 0,C 180,E1 -9688.078,E2 -9688.078} C_VEL
LIN {X 0,Y 425.315,Z 233.985,A -85,B 0,C 180,E1 -9691.373,E2 -9691.373} C_VEL
LIN {X 0,Y 425.276,Z 233.999,A -85,B 0,C 180,E1 -9694.559,E2 -9694.559} C_VEL
LIN {X 0,Y 425.302,Z 234.003,A -85,B 0,C 180,E1 -9697.725,E2 -9697.725} C_VEL
LIN {X 0,Y 425.35,Z 234.001,A -85,B 0,C 180,E1 -9700.709,E2 -9700.709} C_VEL
LIN {X 0,Y 425.375,Z 233.974,A -85,B 0,C 180,E1 -9703.693,E2 -9703.693} C_VEL
LIN {X 0,Y 425.42,Z 233.985,A -85,B 0,C 180,E1 -9707.603,E2 -9707.603} C_VEL
LIN {X 0,Y 425.435,Z 233.992,A -85,B 0,C 180,E1 -9711.454,E2 -9711.454} C_VEL
LIN {X 0,Y 425.549,Z 233.966,A -85,B 0,C 180,E1 -9714.318,E2 -9714.318} C_VEL
LIN {X 0,Y 425.569,Z 233.952,A -85,B 0,C 180,E1 -9718.112,E2 -9718.112} C_VEL
LIN {X 0,Y 425.698,Z 233.949,A -85,B 0,C 180,E1 -9720.004,E2 -9720.004} C_VEL
LIN {X 0,Y 425.544,Z 233.972,A -85,B 0,C 180,E1 -9722.844,E2 -9722.844} C_VEL
LIN {X 0,Y 425.541,Z 233.978,A -85,B 0,C 180,E1 -9725.691,E2 -9725.691} C_VEL
LIN {X 0,Y 425.437,Z 233.973,A -85,B 0,C 180,E1 -9728.554,E2 -9728.554} C_VEL
LIN {X 0,Y 425.414,Z 233.987,A -85,B 0,C 180,E1 -9732.405,E2 -9732.405} C_VEL
LIN {X 0,Y 425.392,Z 233.999,A -85,B 0,C 180,E1 -9736.315,E2 -9736.315} C_VEL
LIN {X 0,Y 425.333,Z 233.991,A -85,B 0,C 180,E1 -9739.639,E2 -9739.639} C_VEL
LIN {X 0,Y 425.293,Z 233.996,A -85,B 0,C 180,E1 -9742.342,E2 -9742.342} C_VEL
LIN {X 0,Y 425.327,Z 234.006,A -85,B 0,C 180,E1 -9744.66,E2 -9744.66} C_VEL
LIN {X 0,Y 425.352,Z 233.995,A -85,B 0,C 180,E1 -9747.561,E2 -9747.561} C_VEL
LIN {X 0,Y 425.295,Z 234,A -85,B 0,C 180,E1 -9750.819,E2 -9750.819} C_VEL
LIN {X 0,Y 425.299,Z 234.006,A -85,B 0,C 180,E1 -9754.286,E2 -9754.286} C_VEL
LIN {X 0,Y 425.284,Z 234.004,A -85,B 0,C 180,E1 -9757.697,E2 -9757.697} C_VEL
LIN {X 0,Y 425.274,Z 234.008,A -85,B 0,C 180,E1 -9760.52,E2 -9760.52} C_VEL
LIN {X 0,Y 425.264,Z 233.999,A -85,B 0,C 180,E1 -9763.352,E2 -9763.352} C_VEL
LIN {X 0,Y 425.27,Z 233.995,A -85,B 0,C 180,E1 -9766.046,E2 -9766.046} C_VEL
LIN {X 0,Y 425.274,Z 234.006,A -85,B 0,C 180,E1 -9768.622,E2 -9768.622} C_VEL
LIN {X 0,Y 425.29,Z 234.005,A -85,B 0,C 180,E1 -9771.101,E2 -9771.101} C_VEL
LIN {X 0,Y 425.308,Z 234.003,A -85,B 0,C 180,E1 -9774.666,E2 -9774.666} C_VEL
LIN {X 0,Y 425.274,Z 234.011,A -85,B 0,C 180,E1 -9778.074,E2 -9778.074} C_VEL
LIN {X 0,Y 425.341,Z 234.003,A -85,B 0,C 180,E1 -9781.369,E2 -9781.369} C_VEL
LIN {X 0,Y 425.379,Z 234.091,A -85,B 0,C 180,E1 -9784.035,E2 -9784.035} C_VEL
LIN {X 0,Y 426.511,Z 239.927,A -85,B 0,C 180,E1 -9785.388,E2 -9785.388} C_VEL
LIN {X 0,Y 427.75,Z 247.753,A -85,B 0,C 180,E1 -9787.086,E2 -9787.086} C_VEL
LIN {X 0,Y 426.777,Z 264.588,A -85,B 0,C 180,E1 -9790.521,E2 -9790.521} C_VEL
LIN {X 0,Y 426.525,Z 269.39,A -85,B 0,C 180,E1 -9791.464,E2 -9791.464} C_VEL
LIN {X 0,Y 427.218,Z 274.402,A -85,B 0,C 180,E1 -9791.623,E2 -9791.623} C_VEL
LIN {X 0,Y 430.16,Z 293.146,A -85,B 0,C 180,E1 -9792.059,E2 -9792.059} C_VEL
LIN {X 0,Y 429.244,Z 377.708,A -85,B 0,C 180,E1 -9793.503,E2 -9793.503} C_VEL
LIN {X 0,Y 428.783,Z 391.599,A -85,B 0,C 180,E1 -9793.944,E2 -9793.944} C_VEL
LIN {X 0,Y 428.224,Z 404.05,A -85,B 0,C 180,E1 -9794.533,E2 -9794.533} C_VEL
LIN {X 0,Y 427.51,Z 416.754,A -85,B 0,C 180,E1 -9795.36,E2 -9795.36} C_VEL
LIN {X 0,Y 426.881,Z 428.565,A -85,B 0,C 180,E1 -9796.358,E2 -9796.358} C_VEL
LIN {X 0,Y 426.291,Z 438.213,A -85,B 0,C 180,E1 -9797.383,E2 -9797.383} C_VEL
LIN {X 0,Y 425.643,Z 447.362,A -85,B 0,C 180,E1 -9798.572,E2 -9798.572} C_VEL
LIN {X 0,Y 425.083,Z 456.278,A -85,B 0,C 180,E1 -9800.003,E2 -9800.003} C_VEL
LIN {X 0,Y 424.672,Z 463.428,A -85,B 0,C 180,E1 -9801.435,E2 -9801.435} C_VEL
LIN {X 0,Y 424.368,Z 469.119,A -85,B 0,C 180,E1 -9802.865,E2 -9802.865} C_VEL
LIN {X 0,Y 424.216,Z 473.597,A -85,B 0,C 180,E1 -9804.296,E2 -9804.296} C_VEL
LIN {X 0,Y 424.21,Z 475.957,A -85,B 0,C 180,E1 -9805.249,E2 -9805.249} C_VEL
LIN {X 0,Y 424.086,Z 477.884,A -85,B 0,C 180,E1 -9806.199,E2 -9806.199} C_VEL
LIN {X 0,Y 424.09,Z 479.382,A -85,B 0,C 180,E1 -9807.151,E2 -9807.151} C_VEL
LIN {X 0,Y 424.126,Z 480.432,A -85,B 0,C 180,E1 -9808.101,E2 -9808.101} C_VEL
LIN {X 0,Y 424.066,Z 481.362,A -85,B 0,C 180,E1 -9810,E2 -9810} C_VEL
LIN {X 0,Y 424.073,Z 481.239,A -85,B 0,C 180,E1 -9810.95,E2 -9810.95} C_VEL
LIN {X 0,Y 424.126,Z 480.685,A -85,B 0,C 180,E1 -9811.899,E2 -9811.899} C_VEL
LIN {X 0,Y 424.086,Z 478.405,A -85,B 0,C 180,E1 -9813.801,E2 -9813.801} C_VEL
LIN {X 0,Y 424.249,Z 475.581,A -85,B 0,C 180,E1 -9815.228,E2 -9815.228} C_VEL
LIN {X 0,Y 424.317,Z 471.738,A -85,B 0,C 180,E1 -9816.658,E2 -9816.658} C_VEL
LIN {X 0,Y 424.599,Z 466.776,A -85,B 0,C 180,E1 -9818.088,E2 -9818.088} C_VEL
LIN {X 0,Y 425.025,Z 460.553,A -85,B 0,C 180,E1 -9819.518,E2 -9819.518} C_VEL
LIN {X 0,Y 425.554,Z 452.792,A -85,B 0,C 180,E1 -9820.948,E2 -9820.948} C_VEL
LIN {X 0,Y 426.359,Z 443.101,A -85,B 0,C 180,E1 -9822.374,E2 -9822.374} C_VEL
LIN {X 0,Y 427.043,Z 433.653,A -85,B 0,C 180,E1 -9823.501,E2 -9823.501} C_VEL
LIN {X 0,Y 427.696,Z 423.196,A -85,B 0,C 180,E1 -9824.513,E2 -9824.513} C_VEL
LIN {X 0,Y 428.563,Z 410.695,A -85,B 0,C 180,E1 -9825.455,E2 -9825.455} C_VEL
LIN {X 0,Y 429.258,Z 398.37,A -85,B 0,C 180,E1 -9826.161,E2 -9826.161} C_VEL
LIN {X 0,Y 429.896,Z 385.266,A -85,B 0,C 180,E1 -9826.686,E2 -9826.686} C_VEL
LIN {X 0,Y 430.222,Z 372.712,A -85,B 0,C 180,E1 -9827.009,E2 -9827.009} C_VEL
LIN {X 0,Y 431.145,Z 292.527,A -85,B 0,C 180,E1 -9828.381,E2 -9828.381} C_VEL
LIN {X 0,Y 427.065,Z 269.853,A -85,B 0,C 180,E1 -9829.009,E2 -9829.009} C_VEL
LIN {X 0,Y 427.034,Z 268.227,A -85,B 0,C 180,E1 -9829.218,E2 -9829.218} C_VEL
LIN {X 0,Y 428.105,Z 251.372,A -85,B 0,C 180,E1 -9832.693,E2 -9832.693} C_VEL
LIN {X 0,Y 428.088,Z 247.772,A -85,B 0,C 180,E1 -9833.461,E2 -9833.461} C_VEL
LIN {X 0,Y 425.723,Z 235.854,A -85,B 0,C 180,E1 -9836.206,E2 -9836.206} C_VEL
LIN {X 0,Y 425.365,Z 234.031,A -85,B 0,C 180,E1 -9836.714,E2 -9836.714} C_VEL
LIN {X 0,Y 425.302,Z 234.009,A -85,B 0,C 180,E1 -9839.719,E2 -9839.719} C_VEL
LIN {X 0,Y 425.295,Z 234.002,A -85,B 0,C 180,E1 -9843.047,E2 -9843.047} C_VEL
LIN {X 0,Y 425.293,Z 234.005,A -85,B 0,C 180,E1 -9845.927,E2 -9845.927} C_VEL
LIN {X 0,Y 425.273,Z 234.004,A -85,B 0,C 180,E1 -9849.036,E2 -9849.036} C_VEL
LIN {X 0,Y 425.281,Z 234.002,A -85,B 0,C 180,E1 -9852.652,E2 -9852.652} C_VEL
LIN {X 0,Y 425.273,Z 234.01,A -85,B 0,C 180,E1 -9856.042,E2 -9856.042} C_VEL
LIN {X 0,Y 425.277,Z 234.005,A -85,B 0,C 180,E1 -9858.618,E2 -9858.618} C_VEL
LIN {X 0,Y 425.292,Z 234.005,A -85,B 0,C 180,E1 -9861.097,E2 -9861.097} C_VEL
LIN {X 0,Y 425.306,Z 234.006,A -85,B 0,C 180,E1 -9864.661,E2 -9864.661} C_VEL
LIN {X 0,Y 425.273,Z 234.004,A -85,B 0,C 180,E1 -9868.07,E2 -9868.07} C_VEL
LIN {X 0,Y 425.315,Z 234.001,A -85,B 0,C 180,E1 -9871.363,E2 -9871.363} C_VEL
LIN {X 0,Y 425.269,Z 234.009,A -85,B 0,C 180,E1 -9874.55,E2 -9874.55} C_VEL
LIN {X 0,Y 425.301,Z 234.006,A -85,B 0,C 180,E1 -9877.727,E2 -9877.727} C_VEL
LIN {X 0,Y 425.37,Z 233.991,A -85,B 0,C 180,E1 -9880.701,E2 -9880.701} C_VEL
LIN {X 0,Y 425.396,Z 233.99,A -85,B 0,C 180,E1 -9883.685,E2 -9883.685} C_VEL
LIN {X 0,Y 425.418,Z 233.994,A -85,B 0,C 180,E1 -9887.595,E2 -9887.595} C_VEL
LIN {X 0,Y 425.411,Z 233.994,A -85,B 0,C 180,E1 -9891.445,E2 -9891.445} C_VEL
LIN {X 0,Y 425.545,Z 233.973,A -85,B 0,C 180,E1 -9894.309,E2 -9894.309} C_VEL
LIN {X 0,Y 425.571,Z 233.969,A -85,B 0,C 180,E1 -9898.103,E2 -9898.103} C_VEL
LIN {X 0,Y 425.698,Z 233.958,A -85,B 0,C 180,E1 -9899.996,E2 -9899.996} C_VEL
LIN {X 0,Y 425.536,Z 233.969,A -85,B 0,C 180,E1 -9902.836,E2 -9902.836} C_VEL
LIN {X 0,Y 425.494,Z 233.977,A -85,B 0,C 180,E1 -9906.512,E2 -9906.512} C_VEL
LIN {X 0,Y 425.393,Z 233.993,A -85,B 0,C 180,E1 -9909.505,E2 -9909.505} C_VEL
LIN {X 0,Y 425.386,Z 233.997,A -85,B 0,C 180,E1 -9912.899,E2 -9912.899} C_VEL
LIN {X 0,Y 425.351,Z 234.002,A -85,B 0,C 180,E1 -9916.6,E2 -9916.6} C_VEL
LIN {X 0,Y 425.316,Z 234.002,A -85,B 0,C 180,E1 -9919.631,E2 -9919.631} C_VEL
LIN {X 0,Y 425.293,Z 234.008,A -85,B 0,C 180,E1 -9923.36,E2 -9923.36} C_VEL
LIN {X 0,Y 425.331,Z 233.992,A -85,B 0,C 180,E1 -9926.839,E2 -9926.839} C_VEL
LIN {X 0,Y 425.271,Z 234.006,A -85,B 0,C 180,E1 -9929.715,E2 -9929.715} C_VEL
LIN {X 0,Y 425.26,Z 234.014,A -85,B 0,C 180,E1 -9933.043,E2 -9933.043} C_VEL
LIN {X 0,Y 425.26,Z 234.012,A -85,B 0,C 180,E1 -9935.924,E2 -9935.924} C_VEL
LIN {X 0,Y 425.288,Z 234.005,A -85,B 0,C 180,E1 -9939.042,E2 -9939.042} C_VEL
LIN {X 0,Y 425.302,Z 234.006,A -85,B 0,C 180,E1 -9942.641,E2 -9942.641} C_VEL
LIN {X 0,Y 425.302,Z 234.009,A -85,B 0,C 180,E1 -9946.049,E2 -9946.049} C_VEL
LIN {X 0,Y 425.33,Z 234.224,A -85,B 0,C 180,E1 -9947.608,E2 -9947.608} C_VEL
LIN {X 0,Y 427.167,Z 242.844,A -85,B 0,C 180,E1 -9949.673,E2 -9949.673} C_VEL
LIN {X 0,Y 427.696,Z 246.71,A -85,B 0,C 180,E1 -9950.552,E2 -9950.552} C_VEL
LIN {X 0,Y 427.161,Z 258.377,A -85,B 0,C 180,E1 -9952.995,E2 -9952.995} C_VEL
LIN {X 0,Y 428.089,Z 263.069,A -85,B 0,C 180,E1 -9953.178,E2 -9953.178} C_VEL
LIN {X 0,Y 431.263,Z 279.645,A -85,B 0,C 180,E1 -9953.636,E2 -9953.636} C_VEL
LIN {X 0,Y 430.167,Z 366.432,A -85,B 0,C 180,E1 -9955.14,E2 -9955.14} C_VEL
LIN {X 0,Y 429.703,Z 380.072,A -85,B 0,C 180,E1 -9955.578,E2 -9955.578} C_VEL
LIN {X 0,Y 429.151,Z 392.387,A -85,B 0,C 180,E1 -9956.165,E2 -9956.165} C_VEL
LIN {X 0,Y 428.467,Z 403.936,A -85,B 0,C 180,E1 -9956.909,E2 -9956.909} C_VEL
LIN {X 0,Y 427.771,Z 415.424,A -85,B 0,C 180,E1 -9957.866,E2 -9957.866} C_VEL
LIN {X 0,Y 426.936,Z 426.299,A -85,B 0,C 180,E1 -9959.001,E2 -9959.001} C_VEL
LIN {X 0,Y 426.281,Z 434.699,A -85,B 0,C 180,E1 -9960.084,E2 -9960.084} C_VEL
LIN {X 0,Y 425.648,Z 443.004,A -85,B 0,C 180,E1 -9961.391,E2 -9961.391} C_VEL
LIN {X 0,Y 425.057,Z 450.702,A -85,B 0,C 180,E1 -9962.89,E2 -9962.89} C_VEL
LIN {X 0,Y 424.627,Z 457.261,A -85,B 0,C 180,E1 -9964.512,E2 -9964.512} C_VEL
LIN {X 0,Y 424.362,Z 462.095,A -85,B 0,C 180,E1 -9966.08,E2 -9966.08} C_VEL
LIN {X 0,Y 424.152,Z 465.57,A -85,B 0,C 180,E1 -9967.598,E2 -9967.598} C_VEL
LIN {X 0,Y 424.053,Z 467.283,A -85,B 0,C 180,E1 -9968.616,E2 -9968.616} C_VEL
LIN {X 0,Y 424.016,Z 468.533,A -85,B 0,C 180,E1 -9969.63,E2 -9969.63} C_VEL
LIN {X 0,Y 423.986,Z 469.391,A -85,B 0,C 180,E1 -9970.859,E2 -9970.859} C_VEL
LIN {X 0,Y 423.948,Z 469.512,A -85,B 0,C 180,E1 -9972.639,E2 -9972.639} C_VEL
LIN {X 0,Y 423.993,Z 468.583,A -85,B 0,C 180,E1 -9974.043,E2 -9974.043} C_VEL
LIN {X 0,Y 424.049,Z 466.556,A -85,B 0,C 180,E1 -9975.605,E2 -9975.605} C_VEL
LIN {X 0,Y 424.23,Z 463.581,A -85,B 0,C 180,E1 -9977.076,E2 -9977.076} C_VEL
LIN {X 0,Y 424.351,Z 461.011,A -85,B 0,C 180,E1 -9978.043,E2 -9978.043} C_VEL
LIN {X 0,Y 423.808,Z 458.801,A -85,B 0,C 180,E1 -9978.779,E2 -9978.779} C_VEL
LIN {X 0,Y 421.16,Z 454.743,A -85,B 0,C 180,E1 -9979.953,E2 -9979.953} C_VEL
LIN {X 0,Y 418.553,Z 450.047,A -85,B 0,C 180,E1 -9981.094,E2 -9981.094} C_VEL
LIN {X 0,Y 418.086,Z 446.792,A -85,B 0,C 180,E1 -9981.771,E2 -9981.771} C_VEL
LIN {X 0,Y 418.64,Z 438.3,A -85,B 0,C 180,E1 -9983.251,E2 -9983.251} C_VEL
LIN {X 0,Y 419.155,Z 429.643,A -85,B 0,C 180,E1 -9984.467,E2 -9984.467} C_VEL
LIN {X 0,Y 419.898,Z 418.941,A -85,B 0,C 180,E1 -9985.68,E2 -9985.68} C_VEL
LIN {X 0,Y 420.624,Z 408.293,A -85,B 0,C 180,E1 -9986.647,E2 -9986.647} C_VEL
LIN {X 0,Y 421.282,Z 396.457,A -85,B 0,C 180,E1 -9987.49,E2 -9987.49} C_VEL
LIN {X 0,Y 421.802,Z 384.163,A -85,B 0,C 180,E1 -9988.15,E2 -9988.15} C_VEL
LIN {X 0,Y 422.209,Z 371.244,A -85,B 0,C 180,E1 -9988.641,E2 -9988.641} C_VEL
LIN {X 0,Y 422.493,Z 357.661,A -85,B 0,C 180,E1 -9988.945,E2 -9988.945} C_VEL
LIN {X 0,Y 423.317,Z 279.29,A -85,B 0,C 180,E1 -9990.282,E2 -9990.282} C_VEL
LIN {X 0,Y 419.726,Z 259.186,A -85,B 0,C 180,E1 -9990.794,E2 -9990.794} C_VEL
LIN {X 0,Y 419.71,Z 257.864,A -85,B 0,C 180,E1 -9990.959,E2 -9990.959} C_VEL
LIN {X 0,Y 420.318,Z 245.901,A -85,B 0,C 180,E1 -9993.595,E2 -9993.595} C_VEL
LIN {X 0,Y 418.492,Z 234.988,A -85,B 0,C 180,E1 -9996.206,E2 -9996.206} C_VEL
LIN {X 0,Y 418.38,Z 234.87,A -85,B 0,C 180,E1 -9999.67,E2 -9999.67} C_VEL
LIN {X 0,Y 418.394,Z 234.868,A -85,B 0,C 180,E1 -10003.059,E2 -10003.059} C_VEL
LIN {X 0,Y 418.292,Z 234.882,A -85,B 0,C 180,E1 -10006.75,E2 -10006.75} C_VEL
LIN {X 0,Y 418.27,Z 234.869,A -85,B 0,C 180,E1 -10009.81,E2 -10009.81} C_VEL
LIN {X 0,Y 418.262,Z 234.885,A -85,B 0,C 180,E1 -10012.734,E2 -10012.734} C_VEL
LIN {X 0,Y 418.229,Z 234.868,A -85,B 0,C 180,E1 -10015.906,E2 -10015.906} C_VEL
LIN {X 0,Y 418.243,Z 234.876,A -85,B 0,C 180,E1 -10019.163,E2 -10019.163} C_VEL
LIN {X 0,Y 418.262,Z 234.888,A -85,B 0,C 180,E1 -10021.391,E2 -10021.391} C_VEL
LIN {X 0,Y 418.239,Z 234.88,A -85,B 0,C 180,E1 -10024.842,E2 -10024.842} C_VEL
LIN {X 0,Y 418.257,Z 234.881,A -85,B 0,C 180,E1 -10028.441,E2 -10028.441} C_VEL
LIN {X 0,Y 418.261,Z 234.871,A -85,B 0,C 180,E1 -10032.23,E2 -10032.23} C_VEL
LIN {X 0,Y 418.255,Z 234.879,A -85,B 0,C 180,E1 -10035.12,E2 -10035.12} C_VEL
LIN {X 0,Y 418.264,Z 234.885,A -85,B 0,C 180,E1 -10037.778,E2 -10037.778} C_VEL
LIN {X 0,Y 418.238,Z 234.868,A -85,B 0,C 180,E1 -10041.564,E2 -10041.564} C_VEL
LIN {X 0,Y 418.233,Z 234.883,A -85,B 0,C 180,E1 -10045.164,E2 -10045.164} C_VEL
LIN {X 0,Y 418.224,Z 234.884,A -85,B 0,C 180,E1 -10047.477,E2 -10047.477} C_VEL
LIN {X 0,Y 418.254,Z 234.867,A -85,B 0,C 180,E1 -10050.898,E2 -10050.898} C_VEL
LIN {X 0,Y 418.251,Z 234.868,A -85,B 0,C 180,E1 -10054.101,E2 -10054.101} C_VEL
LIN {X 0,Y 418.252,Z 234.882,A -85,B 0,C 180,E1 -10057.543,E2 -10057.543} C_VEL
LIN {X 0,Y 418.301,Z 234.875,A -85,B 0,C 180,E1 -10060.371,E2 -10060.371} C_VEL
LIN {X 0,Y 418.303,Z 234.857,A -85,B 0,C 180,E1 -10063.409,E2 -10063.409} C_VEL
LIN {X 0,Y 418.344,Z 234.858,A -85,B 0,C 180,E1 -10066.998,E2 -10066.998} C_VEL
LIN {X 0,Y 418.352,Z 234.868,A -85,B 0,C 180,E1 -10070.334,E2 -10070.334} C_VEL
LIN {X 0,Y 418.488,Z 234.857,A -85,B 0,C 180,E1 -10073.254,E2 -10073.254} C_VEL
LIN {X 0,Y 418.335,Z 234.868,A -85,B 0,C 180,E1 -10075.186,E2 -10075.186} C_VEL
LIN {X 0,Y 418.538,Z 234.827,A -85,B 0,C 180,E1 -10078.08,E2 -10078.08} C_VEL
